// TIA Portal project "BİTİRMEEESON" (V19)

(* hardware
DEVICE "S71500/ET200MP-Station_1"  S7-1500 station
   slot 0: "Profilschiene_0"  6ES7 590-1***0-0AA0
   slot 1: "PLC_1"  CPU 1515-2 PN  6ES7 515-2AM00-0AB0  V1.8
      slot 3: "CPU-Display_1"  6ES7591-1BA00-0AA0
      slot 32768: "PROFINET-Schnittstelle_1"  X1
      slot 33024: "PROFINET interface_1"  X2
   slot 2: "AI 8xU/I/RTD/TC ST_1"  AI 8xU/I/RTD/TC ST  6ES7 531-7KF00-0AB0  V2.0
   slot 3: "AI 8xU/I/RTD/TC ST_2"  AI 8xU/I/RTD/TC ST  6ES7 531-7KF00-0AB0  V2.0
   slot 4: "AI 8xU/I/RTD/TC ST_3"  AI 8xU/I/RTD/TC ST  6ES7 531-7KF00-0AB0  V2.0
   slot 5: "AI 8xU/I/RTD/TC ST_4"  AI 8xU/I/RTD/TC ST  6ES7 531-7KF00-0AB0  V2.0
   slot 6: "DI 16x24VDC BA_1"  DI 16x24VDC BA  6ES7 521-1BH10-0AA0  V1.0
*)

// ===== PLC "PLC_1"  CPU 1515-2 PN =====

VAR_GLOBAL   // PLC tag table "Standard-Variablentabelle"
   "Start_System" AT %I0.0 : Bool;
   "Stop_System" AT %I0.1 : Bool;
   "EmergencyStop" AT %I0.2 : Bool;
   "System" AT %M0.0 : Bool;
   "System_Works_Light" AT %Q0.0 : Bool;
   "System_Not_Working_Light" AT %Q0.1 : Bool;
   "Conveyor1" AT %Q0.2 : Bool;
   "Conveyor2" AT %Q0.3 : Bool;
   "Conveyor3" AT %Q0.4 : Bool;
   "Conveyor4" AT %Q0.5 : Bool;
   "Conveyor5" AT %Q0.6 : Bool;
   "Conveyor6" AT %Q0.7 : Bool;
   "Object_is_Blue" AT %I0.3 : Bool;
   "Object_is_Green" AT %I0.4 : Bool;
   "Blue_So_Left" AT %Q1.0 : Bool;
   "Green_So_Right" AT %Q1.1 : Bool;
   "Mixing_Machine" AT %Q1.2 : Bool;
   "First_Blue_Sensor" AT %I0.5 : Bool;
   "BlueProductConveyor" AT %Q1.3 : Bool;
   "BlueCapConveyor" AT %Q1.4 : Bool;
   "BlueReadyProductConveyor" AT %Q1.5 : Bool;
   "Blue_Product_Sensor" AT %I0.6 : Bool;
   "Blue_Cap_Sensor" AT %I0.7 : Bool;
   "Blue_Product_Positioner" AT %Q1.6 : Bool;
   "Blue_Cap_Positioner" AT %Q1.7 : Bool;
   "Blue_PicknPlace_Grab" AT %Q2.0 : Bool;
   "Blue_PicknPlace_X" AT %Q2.1 : Bool;
   "Blue_PicknPlace_Z" AT %Q2.2 : Bool;
   "Blue_Product_Positioner_Raise" AT %Q2.3 : Bool;
   "Blue_Cap_Emitter" AT %Q2.4 : Bool;
   "Blue_Ready_Sensor" AT %I1.0 : Bool;
   "Blue_Storage_Sensor" AT %I1.1 : Bool;
   "Blue_Roller_Conveyor_1" AT %Q2.5 : Bool;
   "Blue_Roller_Conveyor_2" AT %Q2.6 : Bool;
   "Blue_Roller_Conveyor_3" AT %Q2.7 : Bool;
   "Blue_Roller_Conveyor_4" AT %Q3.0 : Bool;
   "Blue_Roller_Conveyor_5" AT %Q3.1 : Bool;
   "Blue_Roller_Conveyor_6" AT %Q3.2 : Bool;
   "Blue_Ready_Positioner_Clamp" AT %Q3.3 : Bool;
   "Blue_Loading_Conveyor" AT %Q3.4 : Bool;
   "Blue_Box_PicknPlace_X" AT %Q3.5 : Bool;
   "Blue_Box_PicknPlace_Grab" AT %Q3.6 : Bool;
   "Blue_Box_PicknPlace_Z" AT %Q3.7 : Bool;
   "Blue_Conveyor_Blade_1" AT %Q4.0 : Bool;
   "Blue_Conveyor_Blade_2" AT %Q4.1 : Bool;
   "Blue_Box_Emitter" AT %Q4.2 : Bool;
   "Blue_Storage_Start_Button" AT %I1.2 : Bool;
   "Blue_Storage_Stop_Button" AT %I1.3 : Bool;
   "Blue_Storage_Emergency_Button" AT %I1.4 : Bool;
   "Blue_Storage_Start_Button_Main" AT %I1.5 : Bool;
   "Blue_Storage_Stop_Button_Main" AT %I1.6 : Bool;
   "Blue_Storage_Emergency_Button_Main" AT %I1.7 : Bool;
   "Blue_Storage_System" AT %M0.1 : Bool;
   "Blue_Storage_Crane_Left" AT %Q4.3 : Bool;
   "Blue_Storage_Crane_Right" AT %Q4.4 : Bool;
   "Blue_Storage_Crane_Lift" AT %Q4.5 : Bool;
   "Blue_Storage_Start_Button_Light" AT %Q4.6 : Bool;
   "Blue_Storage_Stop_Button_Light" AT %Q4.7 : Bool;
   "Blue_Storage_Start_Button_Main_Light" AT %Q5.0 : Bool;
   "Blue_Storage_Stop_Button_Main_Light" AT %Q5.1 : Bool;
   "Blue_Storage_Reset_Button" AT %I2.0 : Bool;
   "Blue_Storage_Reset_Main_Button" AT %I2.1 : Bool;
   "Blue_Storage_Reset_Button_Light" AT %Q5.2 : Bool;
   "Blue_Storage_Reset_Main_Button_Light" AT %Q5.3 : Bool;
   "Blue_Storage_Crane_Target_Position" AT %QD30 : DInt;
   "Blue_Box_2_Emitter" AT %Q5.4 : Bool;
   "First_Gray_Sensor" AT %I2.2 : Bool;
   "GrayReadyProductConveyor" AT %Q5.5 : Bool;
   "Gray_Cap_Emitter" AT %Q5.6 : Bool;
   "GrayCapConveyor" AT %Q5.7 : Bool;
   "GrayProductConveyor" AT %Q6.0 : Bool;
   "Gray_Product_Sensor" AT %I2.3 : Bool;
   "Gray_Cap_Sensor" AT %I2.4 : Bool;
   "Gray_Product_Positioner" AT %Q6.1 : Bool;
   "Gray_Cap_Positioner" AT %Q6.2 : Bool;
   "Gray_PicknPlace_Grab" AT %Q6.3 : Bool;
   "Gray_PicknPlace_X" AT %Q6.4 : Bool;
   "Gray_PicknPlace_Z" AT %Q6.5 : Bool;
   "Gray_Product_Positioner_Raise" AT %Q6.6 : Bool;
   "Gray_Ready_Sensor" AT %I2.5 : Bool;
   "Gray_Roller_Conveyor_1" AT %Q6.7 : Bool;
   "Gray_Roller_Conveyor_2" AT %Q7.0 : Bool;
   "Gray_Roller_Conveyor_3" AT %Q7.1 : Bool;
   "Gray_Roller_Conveyor_4" AT %Q7.2 : Bool;
   "Gray_Roller_Conveyor_5" AT %Q7.3 : Bool;
   "Gray_Roller_Conveyor_6" AT %Q7.4 : Bool;
   "Gray_Storage_Sensor" AT %I2.6 : Bool;
   "Gray_Loading_Conveyor" AT %Q7.5 : Bool;
   "Gray_Ready_Positioner_Clamp" AT %Q7.6 : Bool;
   "Gray_Box_PicknPlace_X" AT %Q7.7 : Bool;
   "Gray_Box_PicknPlace_Grab" AT %Q8.0 : Bool;
   "Gray_Box_PicknPlace_Z" AT %Q8.1 : Bool;
   "Gray_Box_Emitter" AT %Q8.2 : Bool;
   "Gray_Box_2_Emitter" AT %Q8.3 : Bool;
   "Gray_Conveyor_Blade_1" AT %Q8.4 : Bool;
   "Gray_Conveyor_Blade_2" AT %Q8.5 : Bool;
   "Gray_Storage_Start_Button" AT %I2.7 : Bool;
   "Gray_Storage_Stop_Button" AT %I3.0 : Bool;
   "Gray_Storage_Stop_Button_Main" AT %I3.1 : Bool;
   "Gray_Storage_Emergency_Button" AT %I3.2 : Bool;
   "Gray_Storage_Emergency_Button_Main" AT %I3.3 : Bool;
   "Gray_Storage_System" AT %M0.2 : Bool;
   "Gray_Storage_Start_Button_Main" AT %I3.4 : Bool;
   "Gray_Storage_Reset_Button" AT %I3.5 : Bool;
   "Gray_Storage_Crane_Left" AT %Q8.6 : Bool;
   "Gray_Storage_Reset_Main_Button" AT %I3.6 : Bool;
   "Gray_Storage_Crane_Right" AT %Q8.7 : Bool;
   "Gray_Storage_Crane_Lift" AT %Q9.0 : Bool;
   "Gray_Storage_Start_Button_Light" AT %Q9.1 : Bool;
   "Gray_Storage_Start_Button_Main_Light" AT %Q9.2 : Bool;
   "Gray_Storage_Stop_Button_Light" AT %Q9.3 : Bool;
   "Gray_Storage_Stop_Button_Main_Light" AT %Q9.4 : Bool;
   "Gray_Storage_Reset_Button_Light" AT %Q9.5 : Bool;
   "Gray_Storage_Reset_Main_Button_Light" AT %Q9.6 : Bool;
   "Gray_Storage_Crane_Target_Position" AT %QD34 : DInt;
   "First_Green_Sensor" AT %I3.7 : Bool;
   "GreenReadyProductConveyor" AT %Q9.7 : Bool;
   "Green_Cap_Emitter" AT %Q10.0 : Bool;
   "GreenCapConveyor" AT %Q10.1 : Bool;
   "GreenProductConveyor" AT %Q10.2 : Bool;
   "Green_Product_Positioner" AT %Q10.3 : Bool;
   "Green_Cap_Positioner" AT %Q10.4 : Bool;
   "Green_Product_Sensor" AT %I4.0 : Bool;
   "Green_Cap_Sensor" AT %I4.1 : Bool;
   "Green_PicknPlace_Grab" AT %Q10.5 : Bool;
   "Green_PicknPlace_X" AT %Q10.6 : Bool;
   "Green_PicknPlace_Z" AT %Q10.7 : Bool;
   "Green_Product_Positioner_Raise" AT %Q11.0 : Bool;
   "Green_Ready_Sensor" AT %I4.2 : Bool;
   "Green_Roller_Conveyor_1" AT %Q11.1 : Bool;
   "Green_Roller_Conveyor_2" AT %Q11.2 : Bool;
   "Green_Roller_Conveyor_3" AT %Q11.3 : Bool;
   "Green_Roller_Conveyor_4" AT %Q11.4 : Bool;
   "Green_Roller_Conveyor_5" AT %Q11.5 : Bool;
   "Green_Roller_Conveyor_6" AT %Q11.6 : Bool;
   "Green_Loading_Conveyor" AT %Q11.7 : Bool;
   "Green_Ready_Positioner_Clamp" AT %Q12.0 : Bool;
   "Green_Box_PicknPlace_X" AT %Q12.1 : Bool;
   "Green_Box_PicknPlace_Grab" AT %Q12.2 : Bool;
   "Green_Box_PicknPlace_Z" AT %Q12.3 : Bool;
   "Green_Conveyor_Blade_1" AT %Q12.4 : Bool;
   "Green_Conveyor_Blade_2" AT %Q12.5 : Bool;
   "Green_Box_Emitter" AT %Q12.6 : Bool;
   "Green_Box_2_Emitter" AT %Q12.7 : Bool;
   "Green_Storage_System" AT %M0.3 : Bool;
   "Green_Storage_Start_Button" AT %I4.3 : Bool;
   "Green_Storage_Stop_Button" AT %I4.4 : Bool;
   "Green_Storage_Stop_Button_Main" AT %I4.5 : Bool;
   "Green_Storage_Emergency_Button" AT %I4.6 : Bool;
   "Green_Storage_Emergency_Button_Main" AT %I4.7 : Bool;
   "Green_Storage_Start_Button_Main" AT %I5.0 : Bool;
   "Green_Storage_Reset_Button" AT %I5.1 : Bool;
   "Green_Storage_Reset_Main_Button" AT %I5.2 : Bool;
   "Green_Storage_Crane_Left" AT %Q13.0 : Bool;
   "Green_Storage_Crane_Right" AT %Q13.1 : Bool;
   "Green_Storage_Crane_Lift" AT %Q13.2 : Bool;
   "Green_Storage_Start_Button_Light" AT %Q13.3 : Bool;
   "Green_Storage_Start_Button_Main_Light" AT %Q13.4 : Bool;
   "Green_Storage_Stop_Button_Light" AT %Q13.5 : Bool;
   "Green_Storage_Stop_Button_Main_Light" AT %Q13.6 : Bool;
   "Green_Storage_Reset_Button_Light" AT %Q13.7 : Bool;
   "Green_Storage_Reset_Main_Button_Light" AT %Q14.0 : Bool;
   "Green_Storage_Sensor" AT %I5.3 : Bool;
   "Green_Storage_Crane_Target_Position" AT %QD38 : DInt;
   "MixingCorrectorSensor" AT %I5.4 : Bool;
   "BlueRawEmitter" AT %Q14.1 : Bool;
   "GreenRawEmitter" AT %Q14.2 : Bool;
   "GrayRawEmitter" AT %Q14.3 : Bool;
   "Mixing_Clamp" AT %Q14.4 : Bool;
   "Mixing_Raise" AT %Q14.5 : Bool;
   "Blue_Fill_Valve" AT %QD42 : Real;
   "Blue_Level_Meter" AT %ID30 : DWord;
   "Blue_Liquid_Level" AT %QD56 : DWord;
   "Blue_Norm" AT %MD5 : DWord;
   "Gray_Fill_Valve" AT %QD46 : DWord;
   "Gray_Level_Meter" AT %ID34 : DWord;
   "Gray_Liquid_Level" AT %QD60 : DWord;
   "Gray_Norm" AT %MD6 : DWord;
   "Green_Fill_Valve" AT %QD50 : DWord;
   "Green_Level_Meter" AT %ID38 : DWord;
   "Green_Liquid_Level" AT %QD64 : DWord;
   "Green_Norm" AT %MD7 : DWord;
   "Blue" AT %MW100 : Int;
   "Blue_PID_Flag" AT %M1.0 : Bool;
   "Green_PID_Flag" AT %M1.1 : Bool;
   "Gray_PID_Flag" AT %M1.2 : Bool;
   "Gray" AT %MW104 : Int;
   "Green" AT %MW106 : Int;
   "Blue_Blade_Tank" AT %Q15.2 : Bool;
   "Green_Blade_Tank" AT %Q15.3 : Bool;
   "Gray_Blade_Tank" AT %Q15.4 : Bool;
   "Blue_Base_Vision" AT %I5.5 : Bool;
   "Green_Base_Vision" AT %I5.6 : Bool;
   "Gray_Base_Vision" AT %I5.7 : Bool;
   "BlueDischarge" AT %QD54 : DWord;
   "GreenDischarge" AT %QD58 : DWord;
   "EmitterCycle" AT %M0.4 : Bool;
   "EmittableSituation" AT %M0.5 : Bool;
   "GreenEmit" AT %M0.6 : Bool;
   "GrayEmit" AT %M0.7 : Bool;
   "Conveyor 7" AT %Q14.6 : Bool;
   "Conveyor 8" AT %Q14.7 : Bool;
   "Conveyor 9" AT %Q15.0 : Bool;
   "Conveyor 10" AT %Q15.1 : Bool;
   "Conveyor 11" AT %Q15.5 : Bool;
   "Conveyor 12" AT %Q15.6 : Bool;
   "Conveyor 13" AT %Q15.7 : Bool;
END_VAR

DATA_BLOCK "BrandNewFill_DB"   // DB1
{ S7_Optimized_Access := 'TRUE' }
VERSION : 0.1
// stored: InstanceOfName BrandNewFill
"BrandNewFill"
BEGIN
END_DATA_BLOCK

DATA_BLOCK "Blue_PickPlace_DB"   // DB3
{ S7_Optimized_Access := 'TRUE' }
VERSION : 0.1
// stored: InstanceOfName Blue_PickPlace
"Blue_PickPlace"
BEGIN
END_DATA_BLOCK

DATA_BLOCK "Blue_Storage_Line_DB"   // DB4
{ S7_Optimized_Access := 'TRUE' }
VERSION : 0.1
// stored: InstanceOfName Blue_Storage_Line
"Blue_Storage_Line"
BEGIN
END_DATA_BLOCK

DATA_BLOCK "Blue_Store_DB"   // DB5
{ S7_Optimized_Access := 'TRUE' }
VERSION : 0.1
// stored: InstanceOfName Blue_Store
"Blue_Store"
BEGIN
END_DATA_BLOCK

DATA_BLOCK "Gray_PickPlace_DB"   // DB6
{ S7_Optimized_Access := 'TRUE' }
VERSION : 0.1
// stored: InstanceOfName Gray_PickPlace
"Gray_PickPlace"
BEGIN
END_DATA_BLOCK

DATA_BLOCK "Gray_Storage_Line_DB"   // DB7
{ S7_Optimized_Access := 'TRUE' }
VERSION : 0.1
// stored: InstanceOfName Gray_Storage_Line
"Gray_Storage_Line"
BEGIN
END_DATA_BLOCK

DATA_BLOCK "Gray_Store_DB"   // DB8
{ S7_Optimized_Access := 'TRUE' }
VERSION : 0.1
// stored: InstanceOfName Gray_Store
"Gray_Store"
BEGIN
END_DATA_BLOCK

DATA_BLOCK "Green_PickPlace_DB"   // DB9
{ S7_Optimized_Access := 'TRUE' }
VERSION : 0.1
// stored: InstanceOfName Green_PickPlace
"Green_PickPlace"
BEGIN
END_DATA_BLOCK

DATA_BLOCK "Green_Storage_Line_DB"   // DB10
{ S7_Optimized_Access := 'TRUE' }
VERSION : 0.1
// stored: InstanceOfName Green_Storage_Line
"Green_Storage_Line"
BEGIN
END_DATA_BLOCK

DATA_BLOCK "Green_Store_DB"   // DB11
{ S7_Optimized_Access := 'TRUE' }
VERSION : 0.1
// stored: InstanceOfName Green_Store
"Green_Store"
BEGIN
END_DATA_BLOCK

DATA_BLOCK "MixingCorrector_DB"   // DB108
{ S7_Optimized_Access := 'TRUE' }
VERSION : 0.1
// stored: InstanceOfName MixingCorrector
"MixingCorrector"
BEGIN
END_DATA_BLOCK

// folder: System blocks/Program resources

DATA_BLOCK "TP_BLUEBLADE"   // DB12
{ S7_Optimized_Access := 'TRUE' }
AUTHOR : Simatic
FAMILY : IEC
NAME : IEC_TMR
VERSION : 1.0
// stored: InstanceOfName IEC_TIMER
"IEC_TIMER"
BEGIN
END_DATA_BLOCK

DATA_BLOCK "Blue_Pick&Place"   // DB13
{ S7_Optimized_Access := 'TRUE' }
AUTHOR : Simatic
FAMILY : IEC
NAME : IEC_TMR
VERSION : 1.0
// stored: InstanceOfName IEC_TIMER
"IEC_TIMER"
BEGIN
END_DATA_BLOCK

DATA_BLOCK "Blue_Pick&Place_Grab"   // DB14
{ S7_Optimized_Access := 'TRUE' }
AUTHOR : Simatic
FAMILY : IEC
NAME : IEC_TMR
VERSION : 1.0
// stored: InstanceOfName IEC_TIMER
"IEC_TIMER"
BEGIN
END_DATA_BLOCK

DATA_BLOCK "Blue_Pick&Place_TON_X"   // DB15
{ S7_Optimized_Access := 'TRUE' }
AUTHOR : Simatic
FAMILY : IEC
NAME : IEC_TMR
VERSION : 1.0
// stored: InstanceOfName IEC_TIMER
"IEC_TIMER"
BEGIN
END_DATA_BLOCK

DATA_BLOCK "Blue_Pick&Place_TP_X"   // DB16
{ S7_Optimized_Access := 'TRUE' }
AUTHOR : Simatic
FAMILY : IEC
NAME : IEC_TMR
VERSION : 1.0
// stored: InstanceOfName IEC_TIMER
"IEC_TIMER"
BEGIN
END_DATA_BLOCK

DATA_BLOCK "Blue_Pick&Place_TON_Z1"   // DB17
{ S7_Optimized_Access := 'TRUE' }
AUTHOR : Simatic
FAMILY : IEC
NAME : IEC_TMR
VERSION : 1.0
// stored: InstanceOfName IEC_TIMER
"IEC_TIMER"
BEGIN
END_DATA_BLOCK

DATA_BLOCK "Blue_Pick&PlaceZ2"   // DB18
{ S7_Optimized_Access := 'TRUE' }
AUTHOR : Simatic
FAMILY : IEC
NAME : IEC_TMR
VERSION : 1.0
// stored: InstanceOfName IEC_TIMER
"IEC_TIMER"
BEGIN
END_DATA_BLOCK

DATA_BLOCK "Blue_Pick&PlaceZ3"   // DB19
{ S7_Optimized_Access := 'TRUE' }
AUTHOR : Simatic
FAMILY : IEC
NAME : IEC_TMR
VERSION : 1.0
// stored: InstanceOfName IEC_TIMER
"IEC_TIMER"
BEGIN
END_DATA_BLOCK

DATA_BLOCK "Blue_Raise"   // DB20
{ S7_Optimized_Access := 'TRUE' }
AUTHOR : Simatic
FAMILY : IEC
NAME : IEC_TMR
VERSION : 1.0
// stored: InstanceOfName IEC_TIMER
"IEC_TIMER"
BEGIN
END_DATA_BLOCK

DATA_BLOCK "Blue_Box_Pick&Place"   // DB21
{ S7_Optimized_Access := 'TRUE' }
AUTHOR : Simatic
FAMILY : IEC
NAME : IEC_TMR
VERSION : 1.0
// stored: InstanceOfName IEC_TIMER
"IEC_TIMER"
BEGIN
END_DATA_BLOCK

DATA_BLOCK "Blue_Box_Pick&Place_TON_Grab"   // DB22
{ S7_Optimized_Access := 'TRUE' }
AUTHOR : Simatic
FAMILY : IEC
NAME : IEC_TMR
VERSION : 1.0
// stored: InstanceOfName IEC_TIMER
"IEC_TIMER"
BEGIN
END_DATA_BLOCK

DATA_BLOCK "GrayConveyor"   // DB23
{ S7_Optimized_Access := 'TRUE' }
AUTHOR : Simatic
FAMILY : IEC
NAME : IEC_TMR
VERSION : 1.0
// stored: InstanceOfName IEC_TIMER
"IEC_TIMER"
BEGIN
END_DATA_BLOCK

DATA_BLOCK "Gray_Pick&Place"   // DB24
{ S7_Optimized_Access := 'TRUE' }
AUTHOR : Simatic
FAMILY : IEC
NAME : IEC_TMR
VERSION : 1.0
// stored: InstanceOfName IEC_TIMER
"IEC_TIMER"
BEGIN
END_DATA_BLOCK

DATA_BLOCK "Blue_Storage_Set_TP"   // DB25
{ S7_Optimized_Access := 'TRUE' }
AUTHOR : Simatic
FAMILY : IEC
NAME : IEC_TMR
VERSION : 1.0
// stored: InstanceOfName IEC_TIMER
"IEC_TIMER"
BEGIN
END_DATA_BLOCK

DATA_BLOCK "Blue_Storage_CTU"   // DB26
{ S7_Optimized_Access := 'TRUE' }
AUTHOR : Simatic
FAMILY : IEC
NAME : CNTR
VERSION : 1.0
// stored: InstanceOfName IEC_COUNTER
"IEC_COUNTER"
BEGIN
END_DATA_BLOCK

DATA_BLOCK "Blue_Storage_CTU_Reset_TON"   // DB27
{ S7_Optimized_Access := 'TRUE' }
AUTHOR : Simatic
FAMILY : IEC
NAME : IEC_TMR
VERSION : 1.0
// stored: InstanceOfName IEC_TIMER
"IEC_TIMER"
BEGIN
END_DATA_BLOCK

DATA_BLOCK "Gray_Pick&Place_Grab"   // DB28
{ S7_Optimized_Access := 'TRUE' }
AUTHOR : Simatic
FAMILY : IEC
NAME : IEC_TMR
VERSION : 1.0
// stored: InstanceOfName IEC_TIMER
"IEC_TIMER"
BEGIN
END_DATA_BLOCK

DATA_BLOCK "Gray_Pick&Place_TON_X"   // DB29
{ S7_Optimized_Access := 'TRUE' }
AUTHOR : Simatic
FAMILY : IEC
NAME : IEC_TMR
VERSION : 1.0
// stored: InstanceOfName IEC_TIMER
"IEC_TIMER"
BEGIN
END_DATA_BLOCK

DATA_BLOCK "Blue_Box_Pick&Place_TON_Z1"   // DB30
{ S7_Optimized_Access := 'TRUE' }
AUTHOR : Simatic
FAMILY : IEC
NAME : IEC_TMR
VERSION : 1.0
// stored: InstanceOfName IEC_TIMER
"IEC_TIMER"
BEGIN
END_DATA_BLOCK

DATA_BLOCK "Blue_Box_Pick&Place_TP_Z"   // DB31
{ S7_Optimized_Access := 'TRUE' }
AUTHOR : Simatic
FAMILY : IEC
NAME : IEC_TMR
VERSION : 1.0
// stored: InstanceOfName IEC_TIMER
"IEC_TIMER"
BEGIN
END_DATA_BLOCK

DATA_BLOCK "Blue_Box_Pick&Place_TON_Z2"   // DB32
{ S7_Optimized_Access := 'TRUE' }
AUTHOR : Simatic
FAMILY : IEC
NAME : IEC_TMR
VERSION : 1.0
// stored: InstanceOfName IEC_TIMER
"IEC_TIMER"
BEGIN
END_DATA_BLOCK

DATA_BLOCK "Blue_Box_Pick&Place_TON_Z3"   // DB33
{ S7_Optimized_Access := 'TRUE' }
AUTHOR : Simatic
FAMILY : IEC
NAME : IEC_TMR
VERSION : 1.0
// stored: InstanceOfName IEC_TIMER
"IEC_TIMER"
BEGIN
END_DATA_BLOCK

DATA_BLOCK "Gray_Pick&Place_TP_X"   // DB34
{ S7_Optimized_Access := 'TRUE' }
AUTHOR : Simatic
FAMILY : IEC
NAME : IEC_TMR
VERSION : 1.0
// stored: InstanceOfName IEC_TIMER
"IEC_TIMER"
BEGIN
END_DATA_BLOCK

DATA_BLOCK "Blue_Box_Pick&Place_X"   // DB35
{ S7_Optimized_Access := 'TRUE' }
AUTHOR : Simatic
FAMILY : IEC
NAME : IEC_TMR
VERSION : 1.0
// stored: InstanceOfName IEC_TIMER
"IEC_TIMER"
BEGIN
END_DATA_BLOCK

DATA_BLOCK "Blue_Box_Pick&Place_TP_Grab"   // DB36
{ S7_Optimized_Access := 'TRUE' }
AUTHOR : Simatic
FAMILY : IEC
NAME : IEC_TMR
VERSION : 1.0
// stored: InstanceOfName IEC_TIMER
"IEC_TIMER"
BEGIN
END_DATA_BLOCK

DATA_BLOCK "Gray_Pick&Place_TON_Z1"   // DB37
{ S7_Optimized_Access := 'TRUE' }
AUTHOR : Simatic
FAMILY : IEC
NAME : IEC_TMR
VERSION : 1.0
// stored: InstanceOfName IEC_TIMER
"IEC_TIMER"
BEGIN
END_DATA_BLOCK

DATA_BLOCK "Gray_Pick&PlaceZ2"   // DB38
{ S7_Optimized_Access := 'TRUE' }
AUTHOR : Simatic
FAMILY : IEC
NAME : IEC_TMR
VERSION : 1.0
// stored: InstanceOfName IEC_TIMER
"IEC_TIMER"
BEGIN
END_DATA_BLOCK

DATA_BLOCK "Gray_Pick&PlaceZ3"   // DB39
{ S7_Optimized_Access := 'TRUE' }
AUTHOR : Simatic
FAMILY : IEC
NAME : IEC_TMR
VERSION : 1.0
// stored: InstanceOfName IEC_TIMER
"IEC_TIMER"
BEGIN
END_DATA_BLOCK

DATA_BLOCK "Gray_Raise"   // DB40
{ S7_Optimized_Access := 'TRUE' }
AUTHOR : Simatic
FAMILY : IEC
NAME : IEC_TMR
VERSION : 1.0
// stored: InstanceOfName IEC_TIMER
"IEC_TIMER"
BEGIN
END_DATA_BLOCK

DATA_BLOCK "GrayCapConvey"   // DB41
{ S7_Optimized_Access := 'TRUE' }
AUTHOR : Simatic
FAMILY : IEC
NAME : IEC_TMR
VERSION : 1.0
// stored: InstanceOfName IEC_TIMER
"IEC_TIMER"
BEGIN
END_DATA_BLOCK

DATA_BLOCK "Gray_Box_Pick&Place"   // DB42
{ S7_Optimized_Access := 'TRUE' }
AUTHOR : Simatic
FAMILY : IEC
NAME : IEC_TMR
VERSION : 1.0
// stored: InstanceOfName IEC_TIMER
"IEC_TIMER"
BEGIN
END_DATA_BLOCK

DATA_BLOCK "Gray_Box_Pick&Place_X"   // DB43
{ S7_Optimized_Access := 'TRUE' }
AUTHOR : Simatic
FAMILY : IEC
NAME : IEC_TMR
VERSION : 1.0
// stored: InstanceOfName IEC_TIMER
"IEC_TIMER"
BEGIN
END_DATA_BLOCK

DATA_BLOCK "Gray_Box_Pick&Place_TON_Grab"   // DB44
{ S7_Optimized_Access := 'TRUE' }
AUTHOR : Simatic
FAMILY : IEC
NAME : IEC_TMR
VERSION : 1.0
// stored: InstanceOfName IEC_TIMER
"IEC_TIMER"
BEGIN
END_DATA_BLOCK

DATA_BLOCK "Gray_Box_Pick&Place_TP_Grab"   // DB45
{ S7_Optimized_Access := 'TRUE' }
AUTHOR : Simatic
FAMILY : IEC
NAME : IEC_TMR
VERSION : 1.0
// stored: InstanceOfName IEC_TIMER
"IEC_TIMER"
BEGIN
END_DATA_BLOCK

DATA_BLOCK "Gray_Box_Pick&Place_TON_Z1"   // DB46
{ S7_Optimized_Access := 'TRUE' }
AUTHOR : Simatic
FAMILY : IEC
NAME : IEC_TMR
VERSION : 1.0
// stored: InstanceOfName IEC_TIMER
"IEC_TIMER"
BEGIN
END_DATA_BLOCK

DATA_BLOCK "Gray_Box_Pick&Place_TP_Z"   // DB47
{ S7_Optimized_Access := 'TRUE' }
AUTHOR : Simatic
FAMILY : IEC
NAME : IEC_TMR
VERSION : 1.0
// stored: InstanceOfName IEC_TIMER
"IEC_TIMER"
BEGIN
END_DATA_BLOCK

DATA_BLOCK "Gray_Box_Pick&Place_TON_Z2"   // DB48
{ S7_Optimized_Access := 'TRUE' }
AUTHOR : Simatic
FAMILY : IEC
NAME : IEC_TMR
VERSION : 1.0
// stored: InstanceOfName IEC_TIMER
"IEC_TIMER"
BEGIN
END_DATA_BLOCK

DATA_BLOCK "Gray_Box_Pick&Place_TON_Z3"   // DB49
{ S7_Optimized_Access := 'TRUE' }
AUTHOR : Simatic
FAMILY : IEC
NAME : IEC_TMR
VERSION : 1.0
// stored: InstanceOfName IEC_TIMER
"IEC_TIMER"
BEGIN
END_DATA_BLOCK

DATA_BLOCK "Gray_Box_XTU"   // DB50
{ S7_Optimized_Access := 'TRUE' }
AUTHOR : Simatic
FAMILY : IEC
NAME : CNTR
VERSION : 1.0
// stored: InstanceOfName IEC_COUNTER
"IEC_COUNTER"
BEGIN
END_DATA_BLOCK

DATA_BLOCK "Gray_Box_TON"   // DB51
{ S7_Optimized_Access := 'TRUE' }
AUTHOR : Simatic
FAMILY : IEC
NAME : IEC_TMR
VERSION : 1.0
// stored: InstanceOfName IEC_TIMER
"IEC_TIMER"
BEGIN
END_DATA_BLOCK

DATA_BLOCK "BlueConveyor"   // DB52
{ S7_Optimized_Access := 'TRUE' }
AUTHOR : Simatic
FAMILY : IEC
NAME : IEC_TMR
VERSION : 1.0
// stored: InstanceOfName IEC_TIMER
"IEC_TIMER"
BEGIN
END_DATA_BLOCK

DATA_BLOCK "BlueCapConvey"   // DB53
{ S7_Optimized_Access := 'TRUE' }
AUTHOR : Simatic
FAMILY : IEC
NAME : IEC_TMR
VERSION : 1.0
// stored: InstanceOfName IEC_TIMER
"IEC_TIMER"
BEGIN
END_DATA_BLOCK

DATA_BLOCK "Blue_Box_TON"   // DB54
{ S7_Optimized_Access := 'TRUE' }
AUTHOR : Simatic
FAMILY : IEC
NAME : IEC_TMR
VERSION : 1.0
// stored: InstanceOfName IEC_TIMER
"IEC_TIMER"
BEGIN
END_DATA_BLOCK

DATA_BLOCK "Blue_Box_XTU"   // DB55
{ S7_Optimized_Access := 'TRUE' }
AUTHOR : Simatic
FAMILY : IEC
NAME : CNTR
VERSION : 1.0
// stored: InstanceOfName IEC_COUNTER
"IEC_COUNTER"
BEGIN
END_DATA_BLOCK

DATA_BLOCK "Blue_Box_TP"   // DB56
{ S7_Optimized_Access := 'TRUE' }
AUTHOR : Simatic
FAMILY : IEC
NAME : IEC_TMR
VERSION : 1.0
// stored: InstanceOfName IEC_TIMER
"IEC_TIMER"
BEGIN
END_DATA_BLOCK

DATA_BLOCK "Gray_Box_TP"   // DB57
{ S7_Optimized_Access := 'TRUE' }
AUTHOR : Simatic
FAMILY : IEC
NAME : IEC_TMR
VERSION : 1.0
// stored: InstanceOfName IEC_TIMER
"IEC_TIMER"
BEGIN
END_DATA_BLOCK

DATA_BLOCK "Gray_Storage_CTU"   // DB58
{ S7_Optimized_Access := 'TRUE' }
AUTHOR : Simatic
FAMILY : IEC
NAME : CNTR
VERSION : 1.0
// stored: InstanceOfName IEC_COUNTER
"IEC_COUNTER"
BEGIN
END_DATA_BLOCK

DATA_BLOCK "Gray_Storage_CTU_Reset_TON"   // DB59
{ S7_Optimized_Access := 'TRUE' }
AUTHOR : Simatic
FAMILY : IEC
NAME : IEC_TMR
VERSION : 1.0
// stored: InstanceOfName IEC_TIMER
"IEC_TIMER"
BEGIN
END_DATA_BLOCK

DATA_BLOCK "Gray_Storage_Set_TP"   // DB60
{ S7_Optimized_Access := 'TRUE' }
AUTHOR : Simatic
FAMILY : IEC
NAME : IEC_TMR
VERSION : 1.0
// stored: InstanceOfName IEC_TIMER
"IEC_TIMER"
BEGIN
END_DATA_BLOCK

DATA_BLOCK "Gray_Storage_Crane_Left_Set"   // DB61
{ S7_Optimized_Access := 'TRUE' }
AUTHOR : Simatic
FAMILY : IEC
NAME : IEC_TMR
VERSION : 1.0
// stored: InstanceOfName IEC_TIMER
"IEC_TIMER"
BEGIN
END_DATA_BLOCK

DATA_BLOCK "Gray_Stacker_Crane_Right_Set_TON"   // DB62
{ S7_Optimized_Access := 'TRUE' }
AUTHOR : Simatic
FAMILY : IEC
NAME : IEC_TMR
VERSION : 1.0
// stored: InstanceOfName IEC_TIMER
"IEC_TIMER"
BEGIN
END_DATA_BLOCK

DATA_BLOCK "Gray_Storage_Crane_Right_Set_TP"   // DB63
{ S7_Optimized_Access := 'TRUE' }
AUTHOR : Simatic
FAMILY : IEC
NAME : IEC_TMR
VERSION : 1.0
// stored: InstanceOfName IEC_TIMER
"IEC_TIMER"
BEGIN
END_DATA_BLOCK

DATA_BLOCK "Gray_Storage_Crane_Lift_TON"   // DB64
{ S7_Optimized_Access := 'TRUE' }
AUTHOR : Simatic
FAMILY : IEC
NAME : IEC_TMR
VERSION : 1.0
// stored: InstanceOfName IEC_TIMER
"IEC_TIMER"
BEGIN
END_DATA_BLOCK

DATA_BLOCK "Gray_Storage_Crane_Lift_TP"   // DB65
{ S7_Optimized_Access := 'TRUE' }
AUTHOR : Simatic
FAMILY : IEC
NAME : IEC_TMR
VERSION : 1.0
// stored: InstanceOfName IEC_TIMER
"IEC_TIMER"
BEGIN
END_DATA_BLOCK

DATA_BLOCK "Gray_Storage_Position_Set"   // DB66
{ S7_Optimized_Access := 'TRUE' }
AUTHOR : Simatic
FAMILY : IEC
NAME : IEC_TMR
VERSION : 1.0
// stored: InstanceOfName IEC_TIMER
"IEC_TIMER"
BEGIN
END_DATA_BLOCK

DATA_BLOCK "Gray_Storage_Position_Reset"   // DB67
{ S7_Optimized_Access := 'TRUE' }
AUTHOR : Simatic
FAMILY : IEC
NAME : IEC_TMR
VERSION : 1.0
// stored: InstanceOfName IEC_TIMER
"IEC_TIMER"
BEGIN
END_DATA_BLOCK

DATA_BLOCK "GreenConveyor"   // DB68
{ S7_Optimized_Access := 'TRUE' }
AUTHOR : Simatic
FAMILY : IEC
NAME : IEC_TMR
VERSION : 1.0
// stored: InstanceOfName IEC_TIMER
"IEC_TIMER"
BEGIN
END_DATA_BLOCK

DATA_BLOCK "Blue_Storage_Crane_Left_Set"   // DB69
{ S7_Optimized_Access := 'TRUE' }
AUTHOR : Simatic
FAMILY : IEC
NAME : IEC_TMR
VERSION : 1.0
// stored: InstanceOfName IEC_TIMER
"IEC_TIMER"
BEGIN
END_DATA_BLOCK

DATA_BLOCK "Green_Pick&Place"   // DB70
{ S7_Optimized_Access := 'TRUE' }
AUTHOR : Simatic
FAMILY : IEC
NAME : IEC_TMR
VERSION : 1.0
// stored: InstanceOfName IEC_TIMER
"IEC_TIMER"
BEGIN
END_DATA_BLOCK

DATA_BLOCK "Blue_Stacker_Crane_Right_Set_TON"   // DB71
{ S7_Optimized_Access := 'TRUE' }
AUTHOR : Simatic
FAMILY : IEC
NAME : IEC_TMR
VERSION : 1.0
// stored: InstanceOfName IEC_TIMER
"IEC_TIMER"
BEGIN
END_DATA_BLOCK

DATA_BLOCK "Blue_Storage_Crane_Right_Set_TP"   // DB72
{ S7_Optimized_Access := 'TRUE' }
AUTHOR : Simatic
FAMILY : IEC
NAME : IEC_TMR
VERSION : 1.0
// stored: InstanceOfName IEC_TIMER
"IEC_TIMER"
BEGIN
END_DATA_BLOCK

DATA_BLOCK "Blue_Storage_Crane_Lift_TON"   // DB73
{ S7_Optimized_Access := 'TRUE' }
AUTHOR : Simatic
FAMILY : IEC
NAME : IEC_TMR
VERSION : 1.0
// stored: InstanceOfName IEC_TIMER
"IEC_TIMER"
BEGIN
END_DATA_BLOCK

DATA_BLOCK "Blue_Storage_Crane_Lift_TP"   // DB74
{ S7_Optimized_Access := 'TRUE' }
AUTHOR : Simatic
FAMILY : IEC
NAME : IEC_TMR
VERSION : 1.0
// stored: InstanceOfName IEC_TIMER
"IEC_TIMER"
BEGIN
END_DATA_BLOCK

DATA_BLOCK "Blue_Storage_Position_Set"   // DB75
{ S7_Optimized_Access := 'TRUE' }
AUTHOR : Simatic
FAMILY : IEC
NAME : IEC_TMR
VERSION : 1.0
// stored: InstanceOfName IEC_TIMER
"IEC_TIMER"
BEGIN
END_DATA_BLOCK

DATA_BLOCK "Blue_Storage_Position_Reset"   // DB76
{ S7_Optimized_Access := 'TRUE' }
AUTHOR : Simatic
FAMILY : IEC
NAME : IEC_TMR
VERSION : 1.0
// stored: InstanceOfName IEC_TIMER
"IEC_TIMER"
BEGIN
END_DATA_BLOCK

DATA_BLOCK "Green_Pick&Place_Grab"   // DB77
{ S7_Optimized_Access := 'TRUE' }
AUTHOR : Simatic
FAMILY : IEC
NAME : IEC_TMR
VERSION : 1.0
// stored: InstanceOfName IEC_TIMER
"IEC_TIMER"
BEGIN
END_DATA_BLOCK

DATA_BLOCK "Green_Pick&Place_TON_X"   // DB78
{ S7_Optimized_Access := 'TRUE' }
AUTHOR : Simatic
FAMILY : IEC
NAME : IEC_TMR
VERSION : 1.0
// stored: InstanceOfName IEC_TIMER
"IEC_TIMER"
BEGIN
END_DATA_BLOCK

DATA_BLOCK "Green_Pick&Place_TP_X"   // DB79
{ S7_Optimized_Access := 'TRUE' }
AUTHOR : Simatic
FAMILY : IEC
NAME : IEC_TMR
VERSION : 1.0
// stored: InstanceOfName IEC_TIMER
"IEC_TIMER"
BEGIN
END_DATA_BLOCK

DATA_BLOCK "Green_Pick&Place_TON_Z1"   // DB80
{ S7_Optimized_Access := 'TRUE' }
AUTHOR : Simatic
FAMILY : IEC
NAME : IEC_TMR
VERSION : 1.0
// stored: InstanceOfName IEC_TIMER
"IEC_TIMER"
BEGIN
END_DATA_BLOCK

DATA_BLOCK "Green_Pick&PlaceZ2"   // DB81
{ S7_Optimized_Access := 'TRUE' }
AUTHOR : Simatic
FAMILY : IEC
NAME : IEC_TMR
VERSION : 1.0
// stored: InstanceOfName IEC_TIMER
"IEC_TIMER"
BEGIN
END_DATA_BLOCK

DATA_BLOCK "Green_Pick&PlaceZ3"   // DB82
{ S7_Optimized_Access := 'TRUE' }
AUTHOR : Simatic
FAMILY : IEC
NAME : IEC_TMR
VERSION : 1.0
// stored: InstanceOfName IEC_TIMER
"IEC_TIMER"
BEGIN
END_DATA_BLOCK

DATA_BLOCK "Green_Raise"   // DB83
{ S7_Optimized_Access := 'TRUE' }
AUTHOR : Simatic
FAMILY : IEC
NAME : IEC_TMR
VERSION : 1.0
// stored: InstanceOfName IEC_TIMER
"IEC_TIMER"
BEGIN
END_DATA_BLOCK

DATA_BLOCK "GreenCapConvey"   // DB84
{ S7_Optimized_Access := 'TRUE' }
AUTHOR : Simatic
FAMILY : IEC
NAME : IEC_TMR
VERSION : 1.0
// stored: InstanceOfName IEC_TIMER
"IEC_TIMER"
BEGIN
END_DATA_BLOCK

DATA_BLOCK "Green_Box_Pick&Place"   // DB85
{ S7_Optimized_Access := 'TRUE' }
AUTHOR : Simatic
FAMILY : IEC
NAME : IEC_TMR
VERSION : 1.0
// stored: InstanceOfName IEC_TIMER
"IEC_TIMER"
BEGIN
END_DATA_BLOCK

DATA_BLOCK "Green_Box_Pick&Place_X"   // DB86
{ S7_Optimized_Access := 'TRUE' }
AUTHOR : Simatic
FAMILY : IEC
NAME : IEC_TMR
VERSION : 1.0
// stored: InstanceOfName IEC_TIMER
"IEC_TIMER"
BEGIN
END_DATA_BLOCK

DATA_BLOCK "Green_Box_Pick&Place_TON_Grab"   // DB87
{ S7_Optimized_Access := 'TRUE' }
AUTHOR : Simatic
FAMILY : IEC
NAME : IEC_TMR
VERSION : 1.0
// stored: InstanceOfName IEC_TIMER
"IEC_TIMER"
BEGIN
END_DATA_BLOCK

DATA_BLOCK "Green_Box_Pick&Place_TP_Grab"   // DB88
{ S7_Optimized_Access := 'TRUE' }
AUTHOR : Simatic
FAMILY : IEC
NAME : IEC_TMR
VERSION : 1.0
// stored: InstanceOfName IEC_TIMER
"IEC_TIMER"
BEGIN
END_DATA_BLOCK

DATA_BLOCK "Green_Box_Pick&Place_TON_Z1"   // DB89
{ S7_Optimized_Access := 'TRUE' }
AUTHOR : Simatic
FAMILY : IEC
NAME : IEC_TMR
VERSION : 1.0
// stored: InstanceOfName IEC_TIMER
"IEC_TIMER"
BEGIN
END_DATA_BLOCK

DATA_BLOCK "Green_Box_Pick&Place_TP_Z"   // DB90
{ S7_Optimized_Access := 'TRUE' }
AUTHOR : Simatic
FAMILY : IEC
NAME : IEC_TMR
VERSION : 1.0
// stored: InstanceOfName IEC_TIMER
"IEC_TIMER"
BEGIN
END_DATA_BLOCK

DATA_BLOCK "Green_Box_Pick&Place_TON_Z2"   // DB91
{ S7_Optimized_Access := 'TRUE' }
AUTHOR : Simatic
FAMILY : IEC
NAME : IEC_TMR
VERSION : 1.0
// stored: InstanceOfName IEC_TIMER
"IEC_TIMER"
BEGIN
END_DATA_BLOCK

DATA_BLOCK "Green_Box_Pick&Place_TON_Z3"   // DB92
{ S7_Optimized_Access := 'TRUE' }
AUTHOR : Simatic
FAMILY : IEC
NAME : IEC_TMR
VERSION : 1.0
// stored: InstanceOfName IEC_TIMER
"IEC_TIMER"
BEGIN
END_DATA_BLOCK

DATA_BLOCK "Green_Box_XTU"   // DB93
{ S7_Optimized_Access := 'TRUE' }
AUTHOR : Simatic
FAMILY : IEC
NAME : CNTR
VERSION : 1.0
// stored: InstanceOfName IEC_COUNTER
"IEC_COUNTER"
BEGIN
END_DATA_BLOCK

DATA_BLOCK "Green_Box_TON"   // DB94
{ S7_Optimized_Access := 'TRUE' }
AUTHOR : Simatic
FAMILY : IEC
NAME : IEC_TMR
VERSION : 1.0
// stored: InstanceOfName IEC_TIMER
"IEC_TIMER"
BEGIN
END_DATA_BLOCK

DATA_BLOCK "Green_Box_TP"   // DB95
{ S7_Optimized_Access := 'TRUE' }
AUTHOR : Simatic
FAMILY : IEC
NAME : IEC_TMR
VERSION : 1.0
// stored: InstanceOfName IEC_TIMER
"IEC_TIMER"
BEGIN
END_DATA_BLOCK

DATA_BLOCK "Green_Storage_CTU"   // DB96
{ S7_Optimized_Access := 'TRUE' }
AUTHOR : Simatic
FAMILY : IEC
NAME : CNTR
VERSION : 1.0
// stored: InstanceOfName IEC_COUNTER
"IEC_COUNTER"
BEGIN
END_DATA_BLOCK

DATA_BLOCK "Green_Storage_CTU_Reset_TON"   // DB97
{ S7_Optimized_Access := 'TRUE' }
AUTHOR : Simatic
FAMILY : IEC
NAME : IEC_TMR
VERSION : 1.0
// stored: InstanceOfName IEC_TIMER
"IEC_TIMER"
BEGIN
END_DATA_BLOCK

DATA_BLOCK "Green_Storage_Set_TP"   // DB98
{ S7_Optimized_Access := 'TRUE' }
AUTHOR : Simatic
FAMILY : IEC
NAME : IEC_TMR
VERSION : 1.0
// stored: InstanceOfName IEC_TIMER
"IEC_TIMER"
BEGIN
END_DATA_BLOCK

DATA_BLOCK "Green_Storage_Crane_Left_Set"   // DB99
{ S7_Optimized_Access := 'TRUE' }
AUTHOR : Simatic
FAMILY : IEC
NAME : IEC_TMR
VERSION : 1.0
// stored: InstanceOfName IEC_TIMER
"IEC_TIMER"
BEGIN
END_DATA_BLOCK

DATA_BLOCK "Green_Stacker_Crane_Right_Set_TON"   // DB100
{ S7_Optimized_Access := 'TRUE' }
AUTHOR : Simatic
FAMILY : IEC
NAME : IEC_TMR
VERSION : 1.0
// stored: InstanceOfName IEC_TIMER
"IEC_TIMER"
BEGIN
END_DATA_BLOCK

DATA_BLOCK "Green_Storage_Crane_Right_Set_TP"   // DB101
{ S7_Optimized_Access := 'TRUE' }
AUTHOR : Simatic
FAMILY : IEC
NAME : IEC_TMR
VERSION : 1.0
// stored: InstanceOfName IEC_TIMER
"IEC_TIMER"
BEGIN
END_DATA_BLOCK

DATA_BLOCK "Green_Storage_Crane_Lift_TON"   // DB102
{ S7_Optimized_Access := 'TRUE' }
AUTHOR : Simatic
FAMILY : IEC
NAME : IEC_TMR
VERSION : 1.0
// stored: InstanceOfName IEC_TIMER
"IEC_TIMER"
BEGIN
END_DATA_BLOCK

DATA_BLOCK "Green_Storage_Crane_Lift_TP"   // DB103
{ S7_Optimized_Access := 'TRUE' }
AUTHOR : Simatic
FAMILY : IEC
NAME : IEC_TMR
VERSION : 1.0
// stored: InstanceOfName IEC_TIMER
"IEC_TIMER"
BEGIN
END_DATA_BLOCK

DATA_BLOCK "Green_Storage_Position_Set"   // DB104
{ S7_Optimized_Access := 'TRUE' }
AUTHOR : Simatic
FAMILY : IEC
NAME : IEC_TMR
VERSION : 1.0
// stored: InstanceOfName IEC_TIMER
"IEC_TIMER"
BEGIN
END_DATA_BLOCK

DATA_BLOCK "Green_Storage_Position_Reset"   // DB105
{ S7_Optimized_Access := 'TRUE' }
AUTHOR : Simatic
FAMILY : IEC
NAME : IEC_TMR
VERSION : 1.0
// stored: InstanceOfName IEC_TIMER
"IEC_TIMER"
BEGIN
END_DATA_BLOCK

DATA_BLOCK "MixClampTP"   // DB106
{ S7_Optimized_Access := 'TRUE' }
AUTHOR : Simatic
FAMILY : IEC
NAME : IEC_TMR
VERSION : 1.0
// stored: InstanceOfName IEC_TIMER
"IEC_TIMER"
BEGIN
END_DATA_BLOCK

DATA_BLOCK "MixRaiseTP"   // DB107
{ S7_Optimized_Access := 'TRUE' }
AUTHOR : Simatic
FAMILY : IEC
NAME : IEC_TMR
VERSION : 1.0
// stored: InstanceOfName IEC_TIMER
"IEC_TIMER"
BEGIN
END_DATA_BLOCK

DATA_BLOCK "TP_GREEN_BLADE"   // DB109
{ S7_Optimized_Access := 'TRUE' }
AUTHOR : Simatic
FAMILY : IEC
NAME : IEC_TMR
VERSION : 1.0
// stored: InstanceOfName IEC_TIMER
"IEC_TIMER"
BEGIN
END_DATA_BLOCK

DATA_BLOCK "TP_GRAY_BLADE"   // DB110
{ S7_Optimized_Access := 'TRUE' }
AUTHOR : Simatic
FAMILY : IEC
NAME : IEC_TMR
VERSION : 1.0
// stored: InstanceOfName IEC_TIMER
"IEC_TIMER"
BEGIN
END_DATA_BLOCK

DATA_BLOCK "TONGREEN"   // DB111
{ S7_Optimized_Access := 'TRUE' }
AUTHOR : Simatic
FAMILY : IEC
NAME : IEC_TMR
VERSION : 1.0
// stored: InstanceOfName IEC_TIMER
"IEC_TIMER"
BEGIN
END_DATA_BLOCK

DATA_BLOCK "TONGRay"   // DB112
{ S7_Optimized_Access := 'TRUE' }
AUTHOR : Simatic
FAMILY : IEC
NAME : IEC_TMR
VERSION : 1.0
// stored: InstanceOfName IEC_TIMER
"IEC_TIMER"
BEGIN
END_DATA_BLOCK

DATA_BLOCK "TONBLUE"   // DB113
{ S7_Optimized_Access := 'TRUE' }
AUTHOR : Simatic
FAMILY : IEC
NAME : IEC_TMR
VERSION : 1.0
// stored: InstanceOfName IEC_TIMER
"IEC_TIMER"
BEGIN
END_DATA_BLOCK

DATA_BLOCK "StarterTimer"   // DB114
{ S7_Optimized_Access := 'TRUE' }
AUTHOR : Simatic
FAMILY : IEC
NAME : IEC_TMR
VERSION : 1.0
// stored: InstanceOfName IEC_TIMER
"IEC_TIMER"
BEGIN
END_DATA_BLOCK

DATA_BLOCK "InitialTimer"   // DB115
{ S7_Optimized_Access := 'TRUE' }
AUTHOR : Simatic
FAMILY : IEC
NAME : IEC_TMR
VERSION : 1.0
// stored: InstanceOfName IEC_TIMER
"IEC_TIMER"
BEGIN
END_DATA_BLOCK

DATA_BLOCK "TPGREENTP"   // DB116
{ S7_Optimized_Access := 'TRUE' }
AUTHOR : Simatic
FAMILY : IEC
NAME : IEC_TMR
VERSION : 1.0
// stored: InstanceOfName IEC_TIMER
"IEC_TIMER"
BEGIN
END_DATA_BLOCK

DATA_BLOCK "TPGrayTP"   // DB117
{ S7_Optimized_Access := 'TRUE' }
AUTHOR : Simatic
FAMILY : IEC
NAME : IEC_TMR
VERSION : 1.0
// stored: InstanceOfName IEC_TIMER
"IEC_TIMER"
BEGIN
END_DATA_BLOCK

DATA_BLOCK "TPBLUETP"   // DB118
{ S7_Optimized_Access := 'TRUE' }
AUTHOR : Simatic
FAMILY : IEC
NAME : IEC_TMR
VERSION : 1.0
// stored: InstanceOfName IEC_TIMER
"IEC_TIMER"
BEGIN
END_DATA_BLOCK

// folder: (top level)

FUNCTION_BLOCK "Blue_PickPlace"   // FB1, LAD
{ S7_Optimized_Access := 'TRUE' }
VERSION : 0.1
   VAR_TEMP   // added for the SCL form of the ladder/FBD networks
      _w1 : Bool;
   END_VAR
BEGIN

REGION Network 1
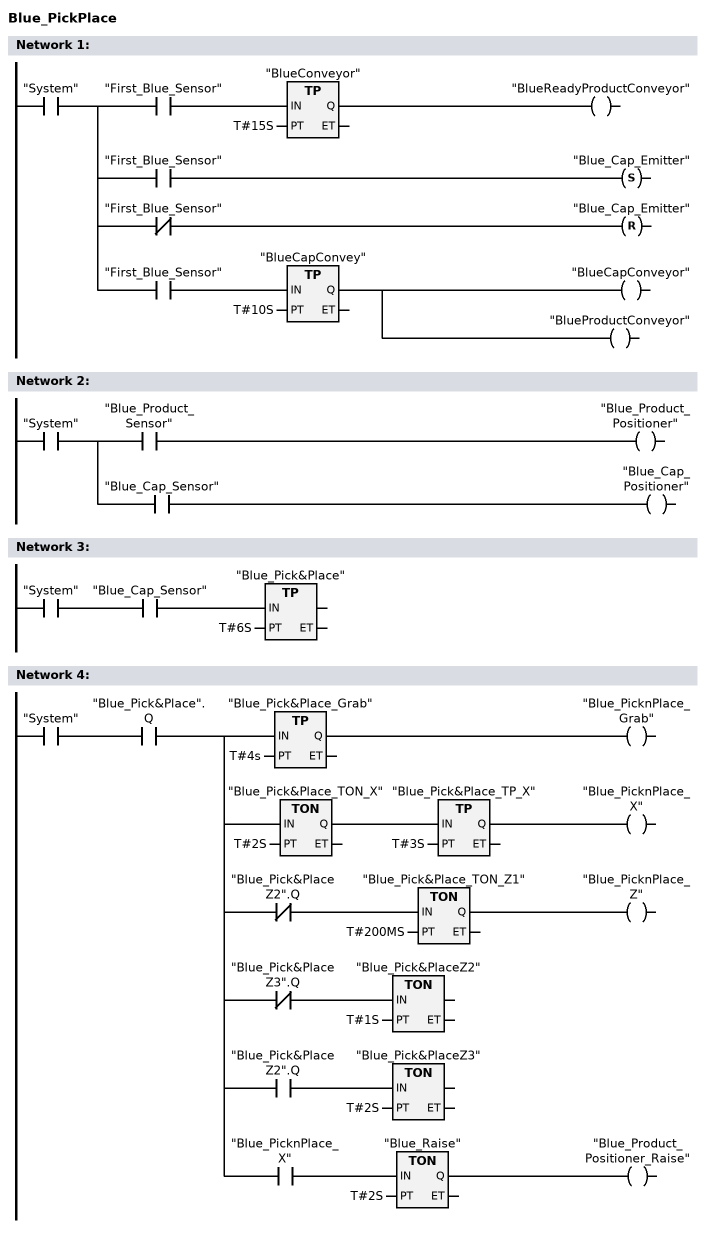
   "BlueConveyor".TP(IN := "System" AND "First_Blue_Sensor", PT := T#15S);
   "BlueReadyProductConveyor" := "BlueConveyor".Q;
   IF "System" AND "First_Blue_Sensor" THEN "Blue_Cap_Emitter" := TRUE; END_IF;
   IF "System" AND NOT "First_Blue_Sensor" THEN "Blue_Cap_Emitter" := FALSE; END_IF;
   "BlueCapConvey".TP(IN := "System" AND "First_Blue_Sensor", PT := T#10S);
   "BlueCapConveyor" := "BlueCapConvey".Q;
   "BlueProductConveyor" := "BlueCapConvey".Q;
END_REGION

REGION Network 2
   RUNG wire#powerrail
      Contact( "System" )
      wire#w1
      Contact( "Blue_Product_Sensor" )
      Coil( "Blue_Product_Positioner" )
   END_RUNG
   RUNG wire#w1
      Contact( "Blue_Cap_Sensor" )
      Coil( "Blue_Cap_Positioner" )
   END_RUNG
   // the same network as SCL:
   "Blue_Product_Positioner" := "System" AND "Blue_Product_Sensor";
   "Blue_Cap_Positioner" := "System" AND "Blue_Cap_Sensor";
END_REGION

REGION Network 3
   "Blue_Pick&Place".TP(IN := "System" AND "Blue_Cap_Sensor", PT := T#6S);
END_REGION

REGION Network 4
   #_w1 := "System" AND "Blue_Pick&Place".Q;
   "Blue_Pick&Place_Grab".TP(IN := #_w1, PT := T#4s);
   "Blue_PicknPlace_Grab" := "Blue_Pick&Place_Grab".Q;
   "Blue_Pick&Place_TON_X".TON(IN := #_w1, PT := T#2S);
   "Blue_Pick&Place_TP_X".TP(IN := "Blue_Pick&Place_TON_X".Q, PT := T#3S);
   "Blue_PicknPlace_X" := "Blue_Pick&Place_TP_X".Q;
   "Blue_Pick&Place_TON_Z1".TON(IN := #_w1 AND NOT "Blue_Pick&PlaceZ2".Q, PT := T#200MS);
   "Blue_PicknPlace_Z" := "Blue_Pick&Place_TON_Z1".Q;
   "Blue_Pick&PlaceZ2".TON(IN := #_w1 AND NOT "Blue_Pick&PlaceZ3".Q, PT := T#1S);
   "Blue_Pick&PlaceZ3".TON(IN := #_w1 AND "Blue_Pick&PlaceZ2".Q, PT := T#2S);
   "Blue_Raise".TON(IN := #_w1 AND "Blue_PicknPlace_X", PT := T#2S);
   "Blue_Product_Positioner_Raise" := "Blue_Raise".Q;
END_REGION
END_FUNCTION_BLOCK

FUNCTION_BLOCK "Blue_Storage_Line"   // FB2, LAD
{ S7_Optimized_Access := 'TRUE' }
VERSION : 0.1
   VAR_TEMP   // added for the SCL form of the ladder/FBD networks
      _w1 : Bool;
   END_VAR
BEGIN

REGION Network 1
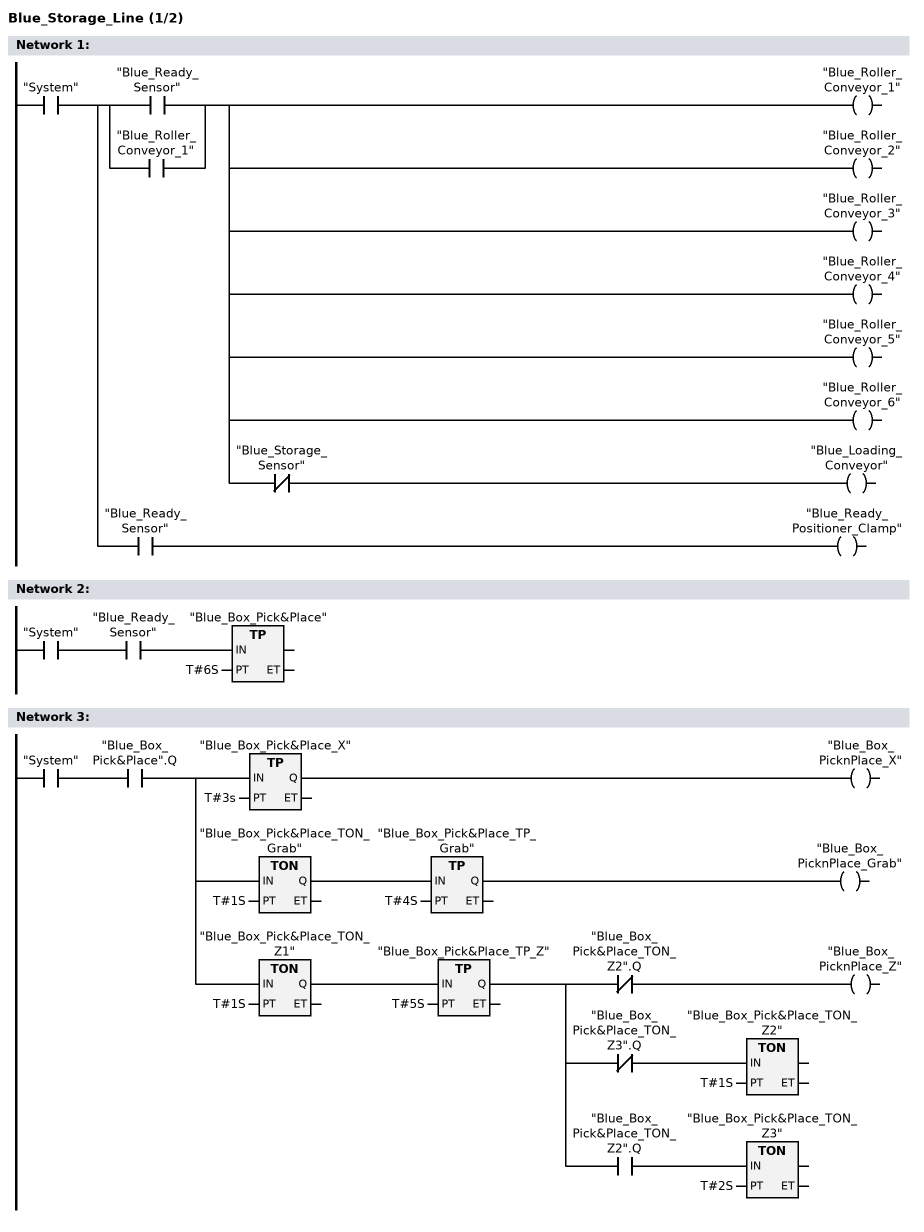
   RUNG wire#powerrail
      Contact( "System" )
      wire#w1
      Contact( "Blue_Ready_Sensor" )
      wire#w2
      Coil( "Blue_Roller_Conveyor_1" )
   END_RUNG
   RUNG wire#w1
      Contact( "Blue_Roller_Conveyor_1" )
   END_RUNG wire#w2
   RUNG wire#w2
      Coil( "Blue_Roller_Conveyor_2" )
   END_RUNG
   RUNG wire#w2
      Coil( "Blue_Roller_Conveyor_3" )
   END_RUNG
   RUNG wire#w2
      Coil( "Blue_Roller_Conveyor_4" )
   END_RUNG
   RUNG wire#w2
      Coil( "Blue_Roller_Conveyor_5" )
   END_RUNG
   RUNG wire#w2
      Coil( "Blue_Roller_Conveyor_6" )
   END_RUNG
   RUNG wire#w2
      I_Contact( "Blue_Storage_Sensor" )
      Coil( "Blue_Loading_Conveyor" )
   END_RUNG
   RUNG wire#w1
      Contact( "Blue_Ready_Sensor" )
      Coil( "Blue_Ready_Positioner_Clamp" )
   END_RUNG
   // the same network as SCL:
   "Blue_Roller_Conveyor_1" := "System" AND ("Blue_Ready_Sensor" OR "Blue_Roller_Conveyor_1");
   "Blue_Roller_Conveyor_2" := "Blue_Roller_Conveyor_1";
   "Blue_Roller_Conveyor_3" := "Blue_Roller_Conveyor_1";
   "Blue_Roller_Conveyor_4" := "Blue_Roller_Conveyor_1";
   "Blue_Roller_Conveyor_5" := "Blue_Roller_Conveyor_1";
   "Blue_Roller_Conveyor_6" := "Blue_Roller_Conveyor_1";
   "Blue_Loading_Conveyor" := "Blue_Roller_Conveyor_1" AND NOT "Blue_Storage_Sensor";
   "Blue_Ready_Positioner_Clamp" := "System" AND "Blue_Ready_Sensor";
END_REGION

REGION Network 2
   "Blue_Box_Pick&Place".TP(IN := "System" AND "Blue_Ready_Sensor", PT := T#6S);
END_REGION

REGION Network 3
   #_w1 := "System" AND "Blue_Box_Pick&Place".Q;
   "Blue_Box_Pick&Place_X".TP(IN := #_w1, PT := T#3s);
   "Blue_Box_PicknPlace_X" := "Blue_Box_Pick&Place_X".Q;
   "Blue_Box_Pick&Place_TON_Grab".TON(IN := #_w1, PT := T#1S);
   "Blue_Box_Pick&Place_TP_Grab".TP(IN := "Blue_Box_Pick&Place_TON_Grab".Q, PT := T#4S);
   "Blue_Box_PicknPlace_Grab" := "Blue_Box_Pick&Place_TP_Grab".Q;
   "Blue_Box_Pick&Place_TON_Z1".TON(IN := #_w1, PT := T#1S);
   "Blue_Box_Pick&Place_TP_Z".TP(IN := "Blue_Box_Pick&Place_TON_Z1".Q, PT := T#5S);
   "Blue_Box_PicknPlace_Z" := "Blue_Box_Pick&Place_TP_Z".Q AND NOT "Blue_Box_Pick&Place_TON_Z2".Q;
   "Blue_Box_Pick&Place_TON_Z2".TON(IN := "Blue_Box_Pick&Place_TP_Z".Q AND NOT "Blue_Box_Pick&Place_TON_Z3".Q,
                           PT := T#1S);
   "Blue_Box_Pick&Place_TON_Z3".TON(IN := "Blue_Box_Pick&Place_TP_Z".Q AND "Blue_Box_Pick&Place_TON_Z2".Q,
                           PT := T#2S);
END_REGION

REGION Network 4
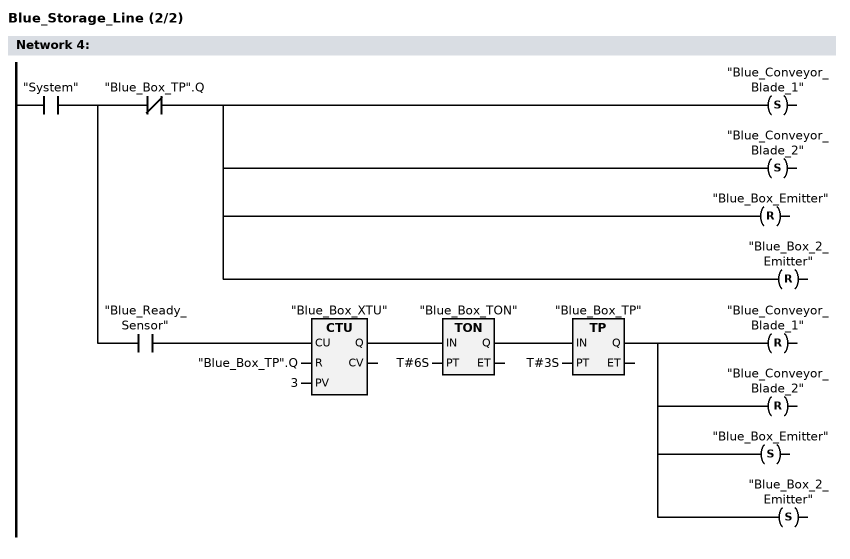
   IF "System" AND NOT "Blue_Box_TP".Q THEN
       "Blue_Conveyor_Blade_1" := TRUE;
       "Blue_Conveyor_Blade_2" := TRUE;
       "Blue_Box_Emitter" := FALSE;
       "Blue_Box_2_Emitter" := FALSE;
   END_IF;
   "Blue_Box_XTU".CTU(CU := "System" AND "Blue_Ready_Sensor", R := "Blue_Box_TP".Q, PV := 3);
   "Blue_Box_TON".TON(IN := "Blue_Box_XTU".Q, PT := T#6S);
   "Blue_Box_TP".TP(IN := "Blue_Box_TON".Q, PT := T#3S);
   IF "Blue_Box_TP".Q THEN
       "Blue_Conveyor_Blade_1" := FALSE;
       "Blue_Conveyor_Blade_2" := FALSE;
       "Blue_Box_Emitter" := TRUE;
       "Blue_Box_2_Emitter" := TRUE;
   END_IF;
END_REGION
END_FUNCTION_BLOCK

FUNCTION_BLOCK "Blue_Store"   // FB3, LAD
{ S7_Optimized_Access := 'TRUE' }
VERSION : 0.1
   VAR_TEMP   // added for the SCL form of the ladder/FBD networks
      _w1 : Bool;
   END_VAR
BEGIN

REGION Network 1
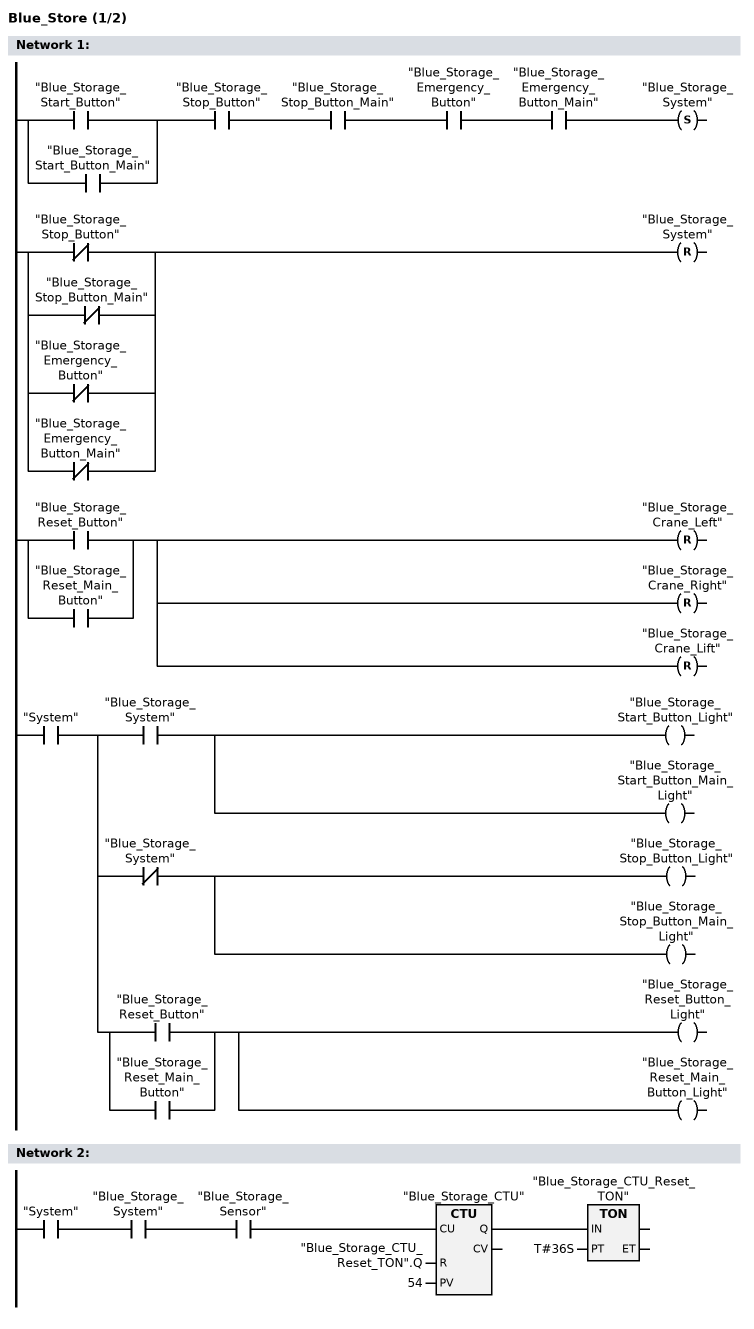
   RUNG wire#powerrail
      Contact( "Blue_Storage_Start_Button" )
      wire#w1
      Contact( "Blue_Storage_Stop_Button" )
      Contact( "Blue_Storage_Stop_Button_Main" )
      Contact( "Blue_Storage_Emergency_Button" )
      Contact( "Blue_Storage_Emergency_Button_Main" )
      S_Coil( "Blue_Storage_System" )
   END_RUNG
   RUNG wire#powerrail
      Contact( "Blue_Storage_Start_Button_Main" )
   END_RUNG wire#w1
   RUNG wire#powerrail
      I_Contact( "Blue_Storage_Stop_Button" )
      wire#w2
      R_Coil( "Blue_Storage_System" )
   END_RUNG
   RUNG wire#powerrail
      I_Contact( "Blue_Storage_Stop_Button_Main" )
   END_RUNG wire#w2
   RUNG wire#powerrail
      I_Contact( "Blue_Storage_Emergency_Button" )
   END_RUNG wire#w2
   RUNG wire#powerrail
      I_Contact( "Blue_Storage_Emergency_Button_Main" )
   END_RUNG wire#w2
   RUNG wire#powerrail
      Contact( "Blue_Storage_Reset_Button" )
      wire#w3
      R_Coil( "Blue_Storage_Crane_Left" )
   END_RUNG
   RUNG wire#powerrail
      Contact( "Blue_Storage_Reset_Main_Button" )
   END_RUNG wire#w3
   RUNG wire#w3
      R_Coil( "Blue_Storage_Crane_Right" )
   END_RUNG
   RUNG wire#w3
      R_Coil( "Blue_Storage_Crane_Lift" )
   END_RUNG
   RUNG wire#powerrail
      Contact( "System" )
      wire#w4
      Contact( "Blue_Storage_System" )
      wire#w5
      Coil( "Blue_Storage_Start_Button_Light" )
   END_RUNG
   RUNG wire#w5
      Coil( "Blue_Storage_Start_Button_Main_Light" )
   END_RUNG
   RUNG wire#w4
      I_Contact( "Blue_Storage_System" )
      wire#w6
      Coil( "Blue_Storage_Stop_Button_Light" )
   END_RUNG
   RUNG wire#w6
      Coil( "Blue_Storage_Stop_Button_Main_Light" )
   END_RUNG
   RUNG wire#w4
      Contact( "Blue_Storage_Reset_Button" )
      wire#w7
      Coil( "Blue_Storage_Reset_Button_Light" )
   END_RUNG
   RUNG wire#w4
      Contact( "Blue_Storage_Reset_Main_Button" )
   END_RUNG wire#w7
   RUNG wire#w7
      Coil( "Blue_Storage_Reset_Main_Button_Light" )
   END_RUNG
   // the same network as SCL:
   IF ("Blue_Storage_Start_Button" OR "Blue_Storage_Start_Button_Main") AND "Blue_Storage_Stop_Button" AND "Blue_Storage_Stop_Button_Main" AND "Blue_Storage_Emergency_Button" AND "Blue_Storage_Emergency_Button_Main" THEN
       "Blue_Storage_System" := TRUE;
   END_IF;
   IF NOT "Blue_Storage_Stop_Button" OR NOT "Blue_Storage_Stop_Button_Main" OR NOT "Blue_Storage_Emergency_Button" OR NOT "Blue_Storage_Emergency_Button_Main" THEN
       "Blue_Storage_System" := FALSE;
   END_IF;
   IF "Blue_Storage_Reset_Button" OR "Blue_Storage_Reset_Main_Button" THEN
       "Blue_Storage_Crane_Left" := FALSE;
       "Blue_Storage_Crane_Right" := FALSE;
       "Blue_Storage_Crane_Lift" := FALSE;
   END_IF;
   "Blue_Storage_Start_Button_Light" := "System" AND "Blue_Storage_System";
   "Blue_Storage_Start_Button_Main_Light" := "Blue_Storage_Start_Button_Light";
   "Blue_Storage_Stop_Button_Light" := "System" AND NOT "Blue_Storage_System";
   "Blue_Storage_Stop_Button_Main_Light" := "Blue_Storage_Stop_Button_Light";
   "Blue_Storage_Reset_Button_Light" := "System" AND ("Blue_Storage_Reset_Button" OR "Blue_Storage_Reset_Main_Button");
   "Blue_Storage_Reset_Main_Button_Light" := "Blue_Storage_Reset_Button_Light";
END_REGION

REGION Network 2
   "Blue_Storage_CTU".CTU(CU := "System" AND "Blue_Storage_System" AND "Blue_Storage_Sensor",
                          R := "Blue_Storage_CTU_Reset_TON".Q,
                          PV := 54);
   "Blue_Storage_CTU_Reset_TON".TON(IN := "Blue_Storage_CTU".Q, PT := T#36S);
END_REGION

REGION Network 3
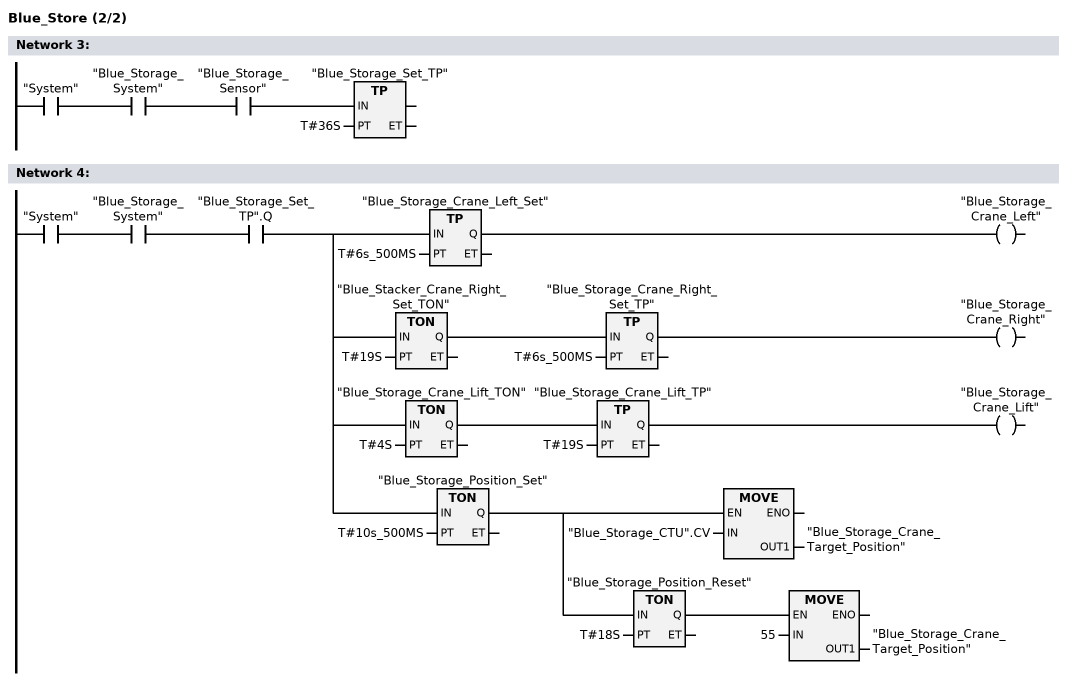
   "Blue_Storage_Set_TP".TP(IN := "System" AND "Blue_Storage_System" AND "Blue_Storage_Sensor", PT := T#36S);
END_REGION

REGION Network 4
   #_w1 := "System" AND "Blue_Storage_System" AND "Blue_Storage_Set_TP".Q;
   "Blue_Storage_Crane_Left_Set".TP(IN := #_w1, PT := T#6s_500MS);
   "Blue_Storage_Crane_Left" := "Blue_Storage_Crane_Left_Set".Q;
   "Blue_Stacker_Crane_Right_Set_TON".TON(IN := #_w1, PT := T#19S);
   "Blue_Storage_Crane_Right_Set_TP".TP(IN := "Blue_Stacker_Crane_Right_Set_TON".Q, PT := T#6s_500MS);
   "Blue_Storage_Crane_Right" := "Blue_Storage_Crane_Right_Set_TP".Q;
   "Blue_Storage_Crane_Lift_TON".TON(IN := #_w1, PT := T#4S);
   "Blue_Storage_Crane_Lift_TP".TP(IN := "Blue_Storage_Crane_Lift_TON".Q, PT := T#19S);
   "Blue_Storage_Crane_Lift" := "Blue_Storage_Crane_Lift_TP".Q;
   "Blue_Storage_Position_Set".TON(IN := #_w1, PT := T#10s_500MS);
   IF "Blue_Storage_Position_Set".Q THEN
       "Blue_Storage_Crane_Target_Position" := "Blue_Storage_CTU".CV;
   END_IF;
   "Blue_Storage_Position_Reset".TON(IN := "Blue_Storage_Position_Set".Q, PT := T#18S);
   IF "Blue_Storage_Position_Reset".Q THEN "Blue_Storage_Crane_Target_Position" := 55; END_IF;
END_REGION
END_FUNCTION_BLOCK

FUNCTION_BLOCK "Gray_PickPlace"   // FB4, LAD
{ S7_Optimized_Access := 'TRUE' }
VERSION : 0.1
   VAR_TEMP   // added for the SCL form of the ladder/FBD networks
      _w1 : Bool;
   END_VAR
BEGIN

REGION Network 1
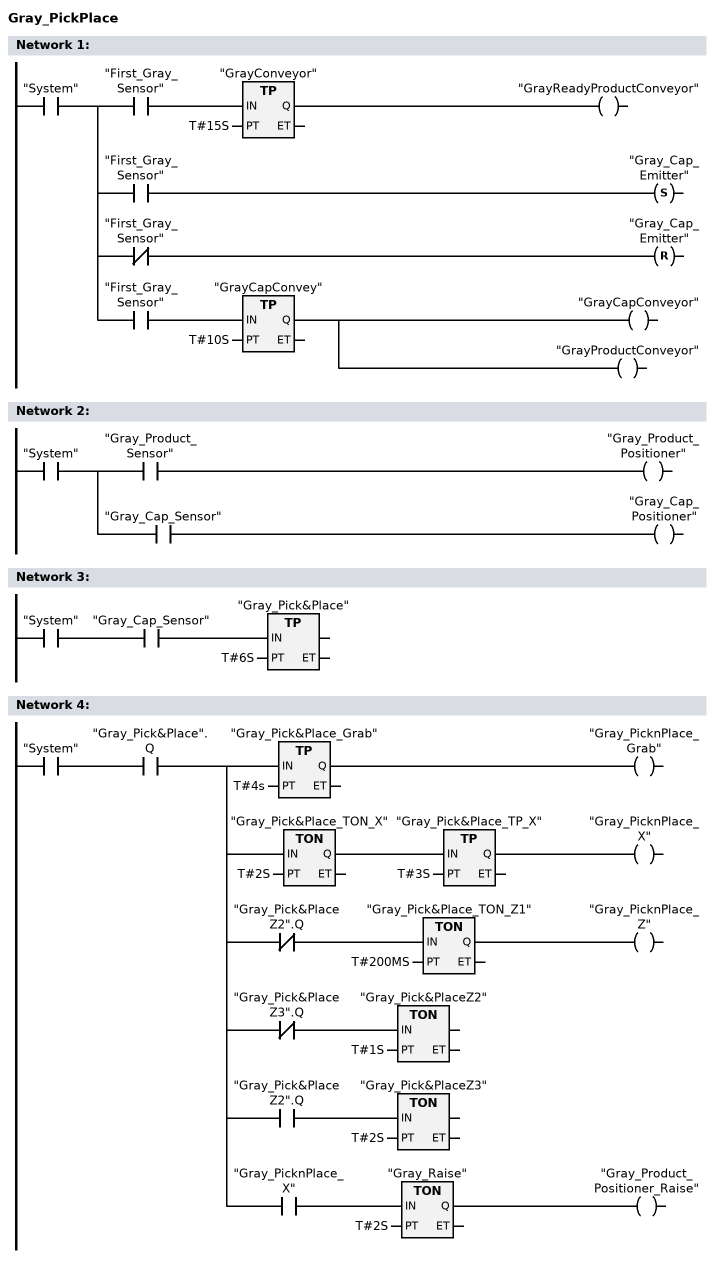
   "GrayConveyor".TP(IN := "System" AND "First_Gray_Sensor", PT := T#15S);
   "GrayReadyProductConveyor" := "GrayConveyor".Q;
   IF "System" AND "First_Gray_Sensor" THEN "Gray_Cap_Emitter" := TRUE; END_IF;
   IF "System" AND NOT "First_Gray_Sensor" THEN "Gray_Cap_Emitter" := FALSE; END_IF;
   "GrayCapConvey".TP(IN := "System" AND "First_Gray_Sensor", PT := T#10S);
   "GrayCapConveyor" := "GrayCapConvey".Q;
   "GrayProductConveyor" := "GrayCapConvey".Q;
END_REGION

REGION Network 2
   RUNG wire#powerrail
      Contact( "System" )
      wire#w1
      Contact( "Gray_Product_Sensor" )
      Coil( "Gray_Product_Positioner" )
   END_RUNG
   RUNG wire#w1
      Contact( "Gray_Cap_Sensor" )
      Coil( "Gray_Cap_Positioner" )
   END_RUNG
   // the same network as SCL:
   "Gray_Product_Positioner" := "System" AND "Gray_Product_Sensor";
   "Gray_Cap_Positioner" := "System" AND "Gray_Cap_Sensor";
END_REGION

REGION Network 3
   "Gray_Pick&Place".TP(IN := "System" AND "Gray_Cap_Sensor", PT := T#6S);
END_REGION

REGION Network 4
   #_w1 := "System" AND "Gray_Pick&Place".Q;
   "Gray_Pick&Place_Grab".TP(IN := #_w1, PT := T#4s);
   "Gray_PicknPlace_Grab" := "Gray_Pick&Place_Grab".Q;
   "Gray_Pick&Place_TON_X".TON(IN := #_w1, PT := T#2S);
   "Gray_Pick&Place_TP_X".TP(IN := "Gray_Pick&Place_TON_X".Q, PT := T#3S);
   "Gray_PicknPlace_X" := "Gray_Pick&Place_TP_X".Q;
   "Gray_Pick&Place_TON_Z1".TON(IN := #_w1 AND NOT "Gray_Pick&PlaceZ2".Q, PT := T#200MS);
   "Gray_PicknPlace_Z" := "Gray_Pick&Place_TON_Z1".Q;
   "Gray_Pick&PlaceZ2".TON(IN := #_w1 AND NOT "Gray_Pick&PlaceZ3".Q, PT := T#1S);
   "Gray_Pick&PlaceZ3".TON(IN := #_w1 AND "Gray_Pick&PlaceZ2".Q, PT := T#2S);
   "Gray_Raise".TON(IN := #_w1 AND "Gray_PicknPlace_X", PT := T#2S);
   "Gray_Product_Positioner_Raise" := "Gray_Raise".Q;
END_REGION
END_FUNCTION_BLOCK

FUNCTION_BLOCK "Gray_Storage_Line"   // FB5, LAD
{ S7_Optimized_Access := 'TRUE' }
VERSION : 0.1
   VAR_TEMP   // added for the SCL form of the ladder/FBD networks
      _w1 : Bool;
   END_VAR
BEGIN

REGION Network 1
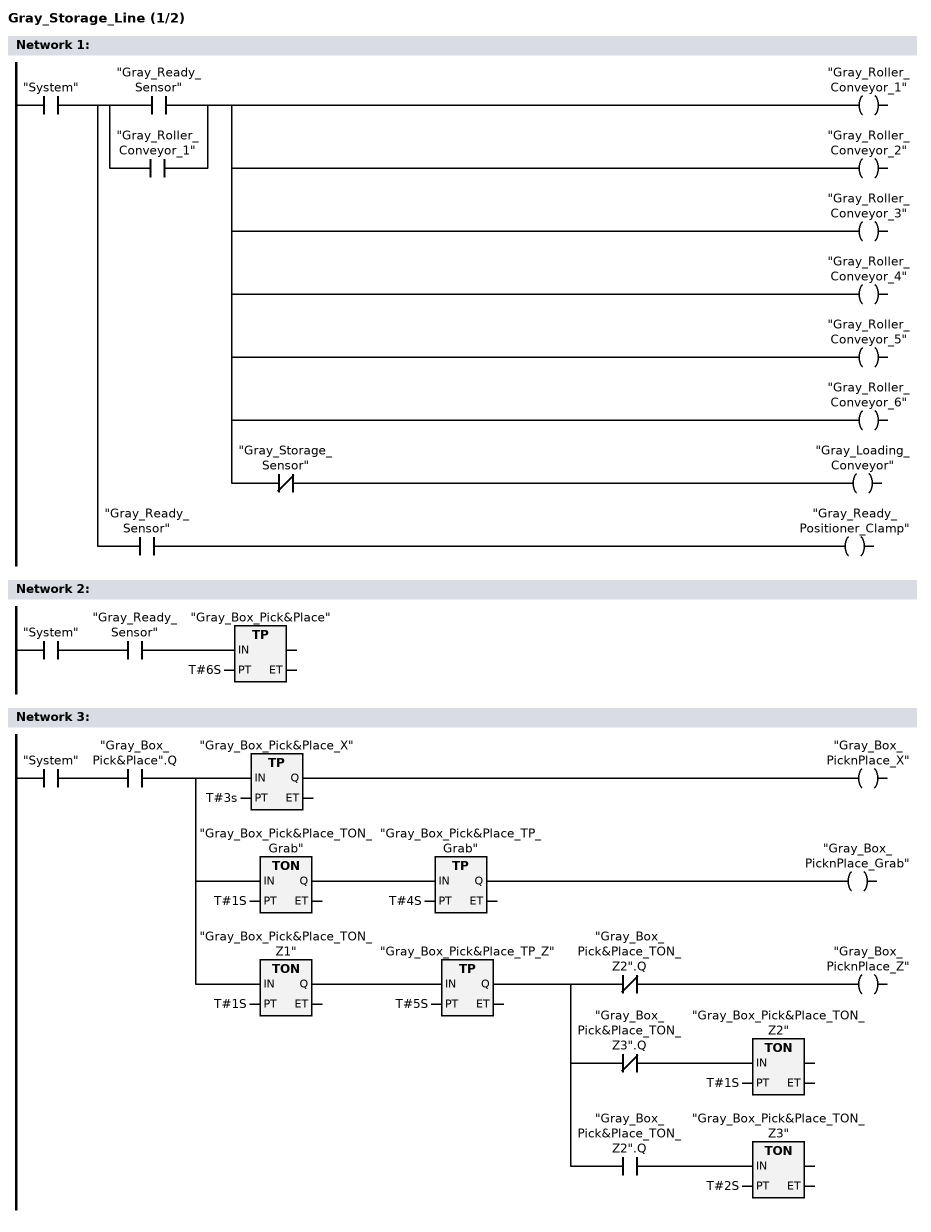
   RUNG wire#powerrail
      Contact( "System" )
      wire#w1
      Contact( "Gray_Ready_Sensor" )
      wire#w2
      Coil( "Gray_Roller_Conveyor_1" )
   END_RUNG
   RUNG wire#w1
      Contact( "Gray_Roller_Conveyor_1" )
   END_RUNG wire#w2
   RUNG wire#w2
      Coil( "Gray_Roller_Conveyor_2" )
   END_RUNG
   RUNG wire#w2
      Coil( "Gray_Roller_Conveyor_3" )
   END_RUNG
   RUNG wire#w2
      Coil( "Gray_Roller_Conveyor_4" )
   END_RUNG
   RUNG wire#w2
      Coil( "Gray_Roller_Conveyor_5" )
   END_RUNG
   RUNG wire#w2
      Coil( "Gray_Roller_Conveyor_6" )
   END_RUNG
   RUNG wire#w2
      I_Contact( "Gray_Storage_Sensor" )
      Coil( "Gray_Loading_Conveyor" )
   END_RUNG
   RUNG wire#w1
      Contact( "Gray_Ready_Sensor" )
      Coil( "Gray_Ready_Positioner_Clamp" )
   END_RUNG
   // the same network as SCL:
   "Gray_Roller_Conveyor_1" := "System" AND ("Gray_Ready_Sensor" OR "Gray_Roller_Conveyor_1");
   "Gray_Roller_Conveyor_2" := "Gray_Roller_Conveyor_1";
   "Gray_Roller_Conveyor_3" := "Gray_Roller_Conveyor_1";
   "Gray_Roller_Conveyor_4" := "Gray_Roller_Conveyor_1";
   "Gray_Roller_Conveyor_5" := "Gray_Roller_Conveyor_1";
   "Gray_Roller_Conveyor_6" := "Gray_Roller_Conveyor_1";
   "Gray_Loading_Conveyor" := "Gray_Roller_Conveyor_1" AND NOT "Gray_Storage_Sensor";
   "Gray_Ready_Positioner_Clamp" := "System" AND "Gray_Ready_Sensor";
END_REGION

REGION Network 2
   "Gray_Box_Pick&Place".TP(IN := "System" AND "Gray_Ready_Sensor", PT := T#6S);
END_REGION

REGION Network 3
   #_w1 := "System" AND "Gray_Box_Pick&Place".Q;
   "Gray_Box_Pick&Place_X".TP(IN := #_w1, PT := T#3s);
   "Gray_Box_PicknPlace_X" := "Gray_Box_Pick&Place_X".Q;
   "Gray_Box_Pick&Place_TON_Grab".TON(IN := #_w1, PT := T#1S);
   "Gray_Box_Pick&Place_TP_Grab".TP(IN := "Gray_Box_Pick&Place_TON_Grab".Q, PT := T#4S);
   "Gray_Box_PicknPlace_Grab" := "Gray_Box_Pick&Place_TP_Grab".Q;
   "Gray_Box_Pick&Place_TON_Z1".TON(IN := #_w1, PT := T#1S);
   "Gray_Box_Pick&Place_TP_Z".TP(IN := "Gray_Box_Pick&Place_TON_Z1".Q, PT := T#5S);
   "Gray_Box_PicknPlace_Z" := "Gray_Box_Pick&Place_TP_Z".Q AND NOT "Gray_Box_Pick&Place_TON_Z2".Q;
   "Gray_Box_Pick&Place_TON_Z2".TON(IN := "Gray_Box_Pick&Place_TP_Z".Q AND NOT "Gray_Box_Pick&Place_TON_Z3".Q,
                           PT := T#1S);
   "Gray_Box_Pick&Place_TON_Z3".TON(IN := "Gray_Box_Pick&Place_TP_Z".Q AND "Gray_Box_Pick&Place_TON_Z2".Q,
                           PT := T#2S);
END_REGION

REGION Network 4
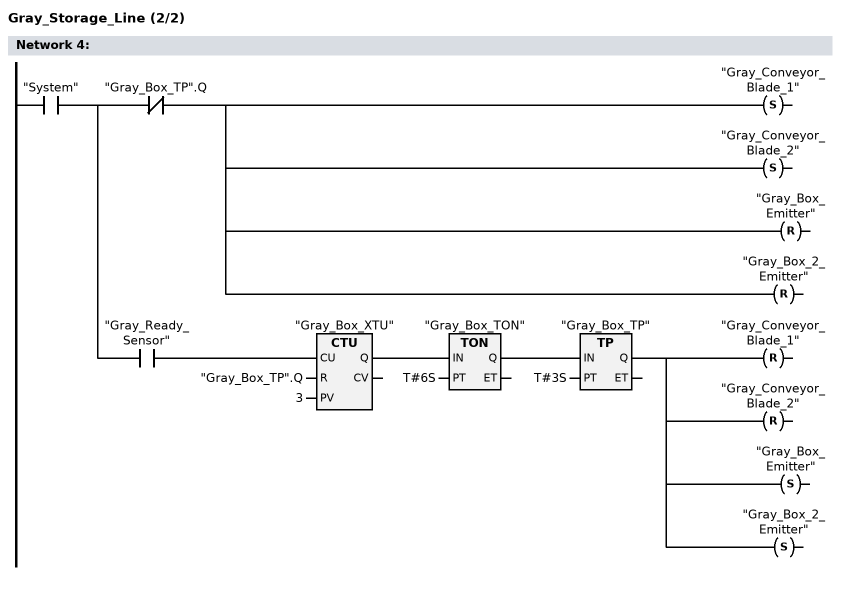
   IF "System" AND NOT "Gray_Box_TP".Q THEN
       "Gray_Conveyor_Blade_1" := TRUE;
       "Gray_Conveyor_Blade_2" := TRUE;
       "Gray_Box_Emitter" := FALSE;
       "Gray_Box_2_Emitter" := FALSE;
   END_IF;
   "Gray_Box_XTU".CTU(CU := "System" AND "Gray_Ready_Sensor", R := "Gray_Box_TP".Q, PV := 3);
   "Gray_Box_TON".TON(IN := "Gray_Box_XTU".Q, PT := T#6S);
   "Gray_Box_TP".TP(IN := "Gray_Box_TON".Q, PT := T#3S);
   IF "Gray_Box_TP".Q THEN
       "Gray_Conveyor_Blade_1" := FALSE;
       "Gray_Conveyor_Blade_2" := FALSE;
       "Gray_Box_Emitter" := TRUE;
       "Gray_Box_2_Emitter" := TRUE;
   END_IF;
END_REGION
END_FUNCTION_BLOCK

FUNCTION_BLOCK "Gray_Store"   // FB6, LAD
{ S7_Optimized_Access := 'TRUE' }
VERSION : 0.1
   VAR_TEMP   // added for the SCL form of the ladder/FBD networks
      _w1 : Bool;
   END_VAR
BEGIN

REGION Network 1
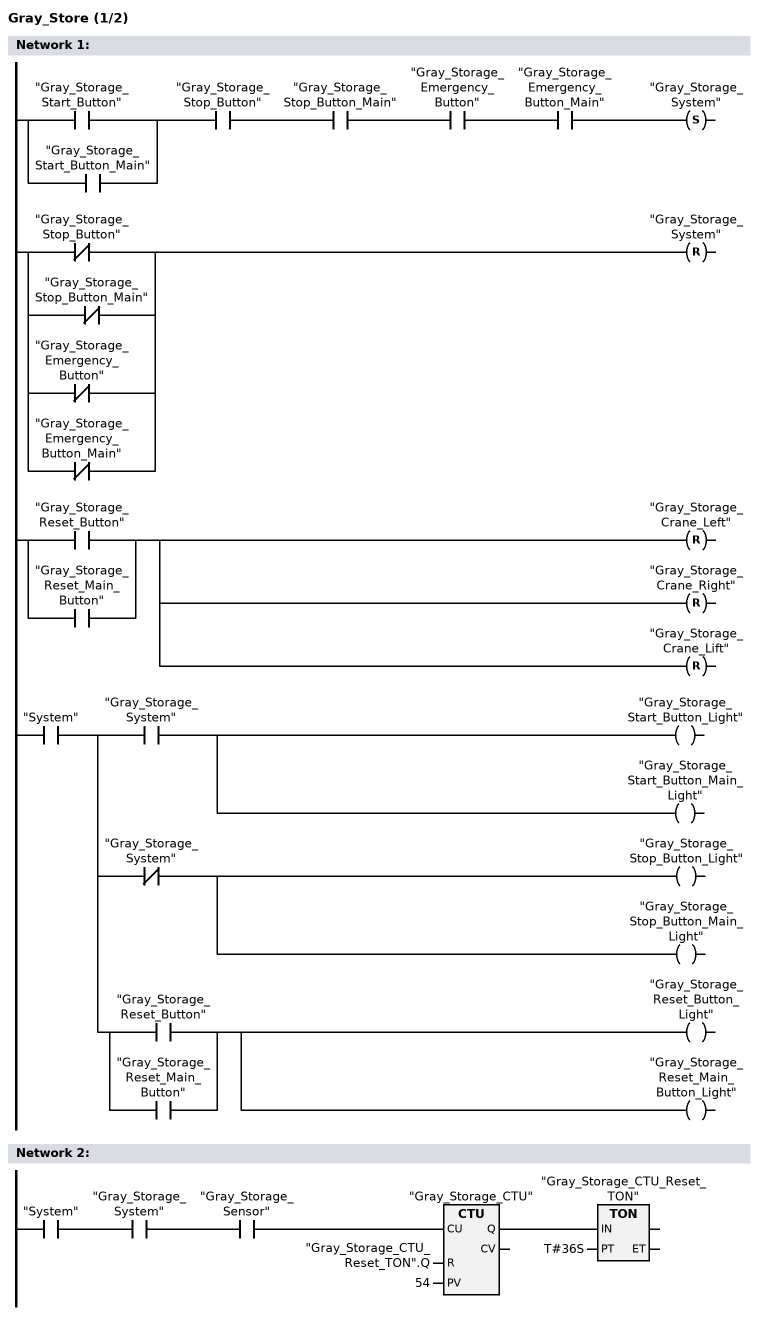
   RUNG wire#powerrail
      Contact( "Gray_Storage_Start_Button" )
      wire#w1
      Contact( "Gray_Storage_Stop_Button" )
      Contact( "Gray_Storage_Stop_Button_Main" )
      Contact( "Gray_Storage_Emergency_Button" )
      Contact( "Gray_Storage_Emergency_Button_Main" )
      S_Coil( "Gray_Storage_System" )
   END_RUNG
   RUNG wire#powerrail
      Contact( "Gray_Storage_Start_Button_Main" )
   END_RUNG wire#w1
   RUNG wire#powerrail
      I_Contact( "Gray_Storage_Stop_Button" )
      wire#w2
      R_Coil( "Gray_Storage_System" )
   END_RUNG
   RUNG wire#powerrail
      I_Contact( "Gray_Storage_Stop_Button_Main" )
   END_RUNG wire#w2
   RUNG wire#powerrail
      I_Contact( "Gray_Storage_Emergency_Button" )
   END_RUNG wire#w2
   RUNG wire#powerrail
      I_Contact( "Gray_Storage_Emergency_Button_Main" )
   END_RUNG wire#w2
   RUNG wire#powerrail
      Contact( "Gray_Storage_Reset_Button" )
      wire#w3
      R_Coil( "Gray_Storage_Crane_Left" )
   END_RUNG
   RUNG wire#powerrail
      Contact( "Gray_Storage_Reset_Main_Button" )
   END_RUNG wire#w3
   RUNG wire#w3
      R_Coil( "Gray_Storage_Crane_Right" )
   END_RUNG
   RUNG wire#w3
      R_Coil( "Gray_Storage_Crane_Lift" )
   END_RUNG
   RUNG wire#powerrail
      Contact( "System" )
      wire#w4
      Contact( "Gray_Storage_System" )
      wire#w5
      Coil( "Gray_Storage_Start_Button_Light" )
   END_RUNG
   RUNG wire#w5
      Coil( "Gray_Storage_Start_Button_Main_Light" )
   END_RUNG
   RUNG wire#w4
      I_Contact( "Gray_Storage_System" )
      wire#w6
      Coil( "Gray_Storage_Stop_Button_Light" )
   END_RUNG
   RUNG wire#w6
      Coil( "Gray_Storage_Stop_Button_Main_Light" )
   END_RUNG
   RUNG wire#w4
      Contact( "Gray_Storage_Reset_Button" )
      wire#w7
      Coil( "Gray_Storage_Reset_Button_Light" )
   END_RUNG
   RUNG wire#w4
      Contact( "Gray_Storage_Reset_Main_Button" )
   END_RUNG wire#w7
   RUNG wire#w7
      Coil( "Gray_Storage_Reset_Main_Button_Light" )
   END_RUNG
   // the same network as SCL:
   IF ("Gray_Storage_Start_Button" OR "Gray_Storage_Start_Button_Main") AND "Gray_Storage_Stop_Button" AND "Gray_Storage_Stop_Button_Main" AND "Gray_Storage_Emergency_Button" AND "Gray_Storage_Emergency_Button_Main" THEN
       "Gray_Storage_System" := TRUE;
   END_IF;
   IF NOT "Gray_Storage_Stop_Button" OR NOT "Gray_Storage_Stop_Button_Main" OR NOT "Gray_Storage_Emergency_Button" OR NOT "Gray_Storage_Emergency_Button_Main" THEN
       "Gray_Storage_System" := FALSE;
   END_IF;
   IF "Gray_Storage_Reset_Button" OR "Gray_Storage_Reset_Main_Button" THEN
       "Gray_Storage_Crane_Left" := FALSE;
       "Gray_Storage_Crane_Right" := FALSE;
       "Gray_Storage_Crane_Lift" := FALSE;
   END_IF;
   "Gray_Storage_Start_Button_Light" := "System" AND "Gray_Storage_System";
   "Gray_Storage_Start_Button_Main_Light" := "Gray_Storage_Start_Button_Light";
   "Gray_Storage_Stop_Button_Light" := "System" AND NOT "Gray_Storage_System";
   "Gray_Storage_Stop_Button_Main_Light" := "Gray_Storage_Stop_Button_Light";
   "Gray_Storage_Reset_Button_Light" := "System" AND ("Gray_Storage_Reset_Button" OR "Gray_Storage_Reset_Main_Button");
   "Gray_Storage_Reset_Main_Button_Light" := "Gray_Storage_Reset_Button_Light";
END_REGION

REGION Network 2
   "Gray_Storage_CTU".CTU(CU := "System" AND "Gray_Storage_System" AND "Gray_Storage_Sensor",
                          R := "Gray_Storage_CTU_Reset_TON".Q,
                          PV := 54);
   "Gray_Storage_CTU_Reset_TON".TON(IN := "Gray_Storage_CTU".Q, PT := T#36S);
END_REGION

REGION Network 3
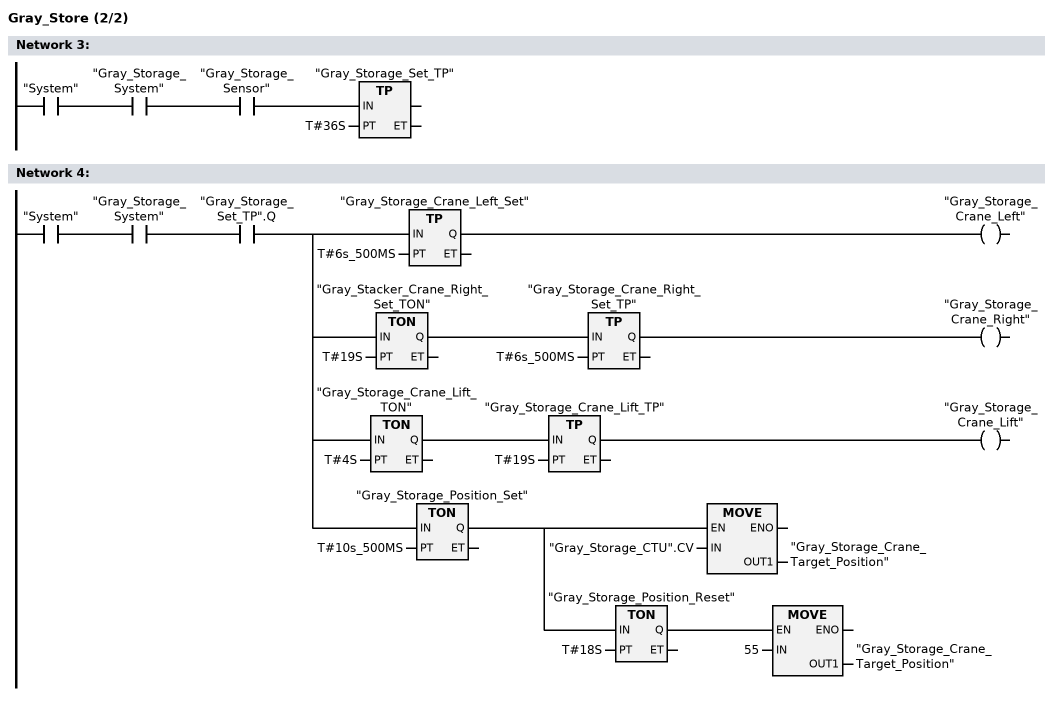
   "Gray_Storage_Set_TP".TP(IN := "System" AND "Gray_Storage_System" AND "Gray_Storage_Sensor", PT := T#36S);
END_REGION

REGION Network 4
   #_w1 := "System" AND "Gray_Storage_System" AND "Gray_Storage_Set_TP".Q;
   "Gray_Storage_Crane_Left_Set".TP(IN := #_w1, PT := T#6s_500MS);
   "Gray_Storage_Crane_Left" := "Gray_Storage_Crane_Left_Set".Q;
   "Gray_Stacker_Crane_Right_Set_TON".TON(IN := #_w1, PT := T#19S);
   "Gray_Storage_Crane_Right_Set_TP".TP(IN := "Gray_Stacker_Crane_Right_Set_TON".Q, PT := T#6s_500MS);
   "Gray_Storage_Crane_Right" := "Gray_Storage_Crane_Right_Set_TP".Q;
   "Gray_Storage_Crane_Lift_TON".TON(IN := #_w1, PT := T#4S);
   "Gray_Storage_Crane_Lift_TP".TP(IN := "Gray_Storage_Crane_Lift_TON".Q, PT := T#19S);
   "Gray_Storage_Crane_Lift" := "Gray_Storage_Crane_Lift_TP".Q;
   "Gray_Storage_Position_Set".TON(IN := #_w1, PT := T#10s_500MS);
   IF "Gray_Storage_Position_Set".Q THEN
       "Gray_Storage_Crane_Target_Position" := "Gray_Storage_CTU".CV;
   END_IF;
   "Gray_Storage_Position_Reset".TON(IN := "Gray_Storage_Position_Set".Q, PT := T#18S);
   IF "Gray_Storage_Position_Reset".Q THEN "Gray_Storage_Crane_Target_Position" := 55; END_IF;
END_REGION
END_FUNCTION_BLOCK

FUNCTION_BLOCK "Green_PickPlace"   // FB7, LAD
{ S7_Optimized_Access := 'TRUE' }
VERSION : 0.1
   VAR_TEMP   // added for the SCL form of the ladder/FBD networks
      _w1 : Bool;
   END_VAR
BEGIN

REGION Network 1
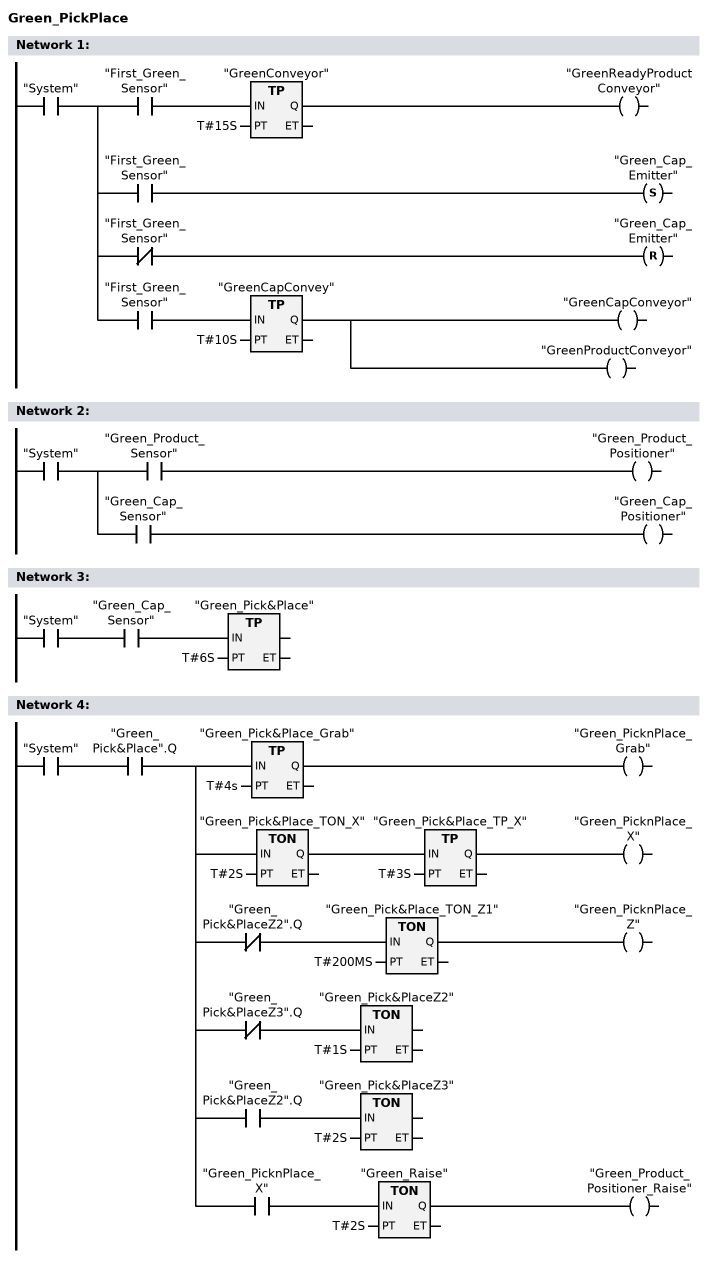
   "GreenConveyor".TP(IN := "System" AND "First_Green_Sensor", PT := T#15S);
   "GreenReadyProductConveyor" := "GreenConveyor".Q;
   IF "System" AND "First_Green_Sensor" THEN "Green_Cap_Emitter" := TRUE; END_IF;
   IF "System" AND NOT "First_Green_Sensor" THEN "Green_Cap_Emitter" := FALSE; END_IF;
   "GreenCapConvey".TP(IN := "System" AND "First_Green_Sensor", PT := T#10S);
   "GreenCapConveyor" := "GreenCapConvey".Q;
   "GreenProductConveyor" := "GreenCapConvey".Q;
END_REGION

REGION Network 2
   RUNG wire#powerrail
      Contact( "System" )
      wire#w1
      Contact( "Green_Product_Sensor" )
      Coil( "Green_Product_Positioner" )
   END_RUNG
   RUNG wire#w1
      Contact( "Green_Cap_Sensor" )
      Coil( "Green_Cap_Positioner" )
   END_RUNG
   // the same network as SCL:
   "Green_Product_Positioner" := "System" AND "Green_Product_Sensor";
   "Green_Cap_Positioner" := "System" AND "Green_Cap_Sensor";
END_REGION

REGION Network 3
   "Green_Pick&Place".TP(IN := "System" AND "Green_Cap_Sensor", PT := T#6S);
END_REGION

REGION Network 4
   #_w1 := "System" AND "Green_Pick&Place".Q;
   "Green_Pick&Place_Grab".TP(IN := #_w1, PT := T#4s);
   "Green_PicknPlace_Grab" := "Green_Pick&Place_Grab".Q;
   "Green_Pick&Place_TON_X".TON(IN := #_w1, PT := T#2S);
   "Green_Pick&Place_TP_X".TP(IN := "Green_Pick&Place_TON_X".Q, PT := T#3S);
   "Green_PicknPlace_X" := "Green_Pick&Place_TP_X".Q;
   "Green_Pick&Place_TON_Z1".TON(IN := #_w1 AND NOT "Green_Pick&PlaceZ2".Q, PT := T#200MS);
   "Green_PicknPlace_Z" := "Green_Pick&Place_TON_Z1".Q;
   "Green_Pick&PlaceZ2".TON(IN := #_w1 AND NOT "Green_Pick&PlaceZ3".Q, PT := T#1S);
   "Green_Pick&PlaceZ3".TON(IN := #_w1 AND "Green_Pick&PlaceZ2".Q, PT := T#2S);
   "Green_Raise".TON(IN := #_w1 AND "Green_PicknPlace_X", PT := T#2S);
   "Green_Product_Positioner_Raise" := "Green_Raise".Q;
END_REGION
END_FUNCTION_BLOCK

FUNCTION_BLOCK "Green_Storage_Line"   // FB8, LAD
{ S7_Optimized_Access := 'TRUE' }
VERSION : 0.1
   VAR_TEMP   // added for the SCL form of the ladder/FBD networks
      _w1 : Bool;
   END_VAR
BEGIN

REGION Network 1
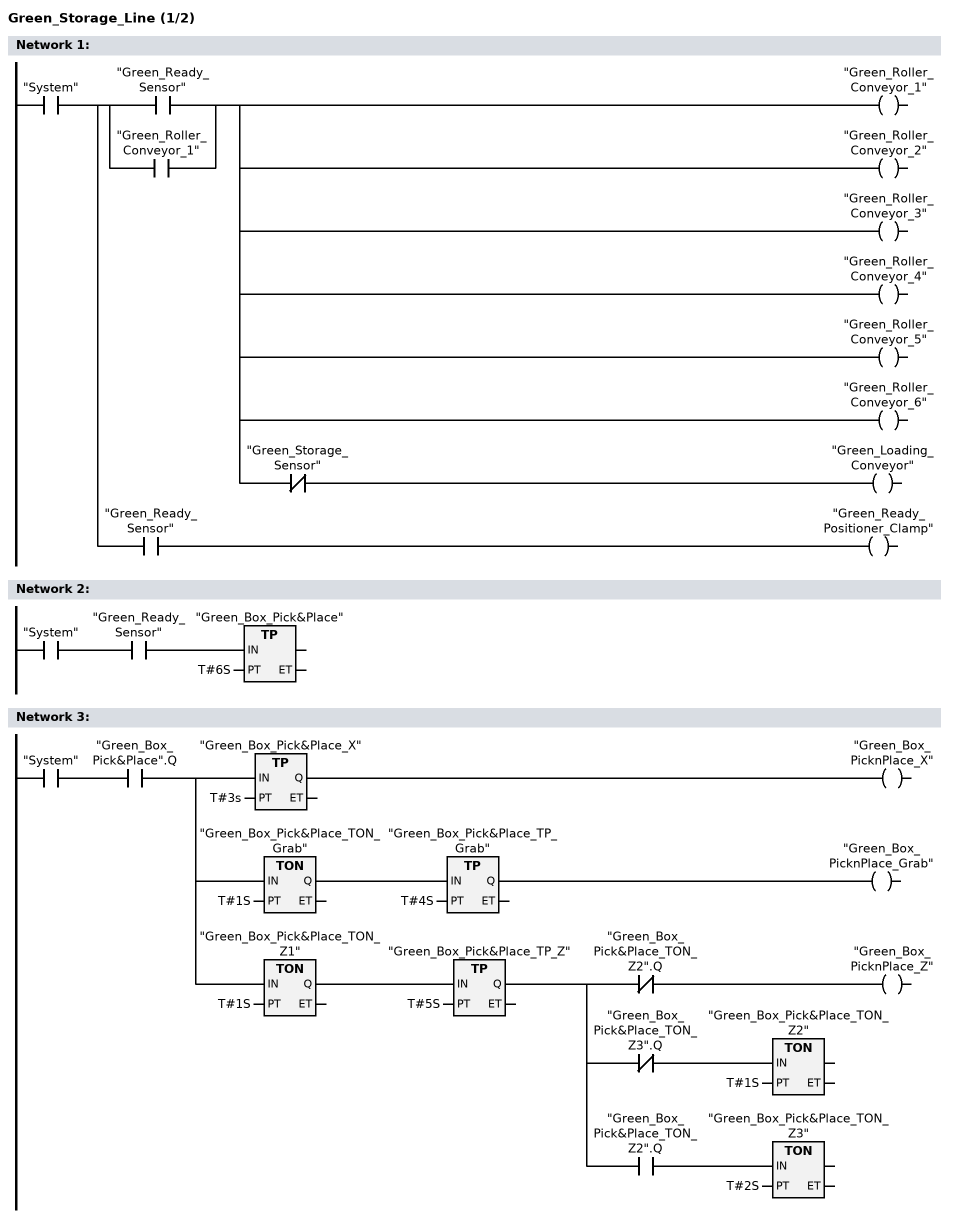
   RUNG wire#powerrail
      Contact( "System" )
      wire#w1
      Contact( "Green_Ready_Sensor" )
      wire#w2
      Coil( "Green_Roller_Conveyor_1" )
   END_RUNG
   RUNG wire#w1
      Contact( "Green_Roller_Conveyor_1" )
   END_RUNG wire#w2
   RUNG wire#w2
      Coil( "Green_Roller_Conveyor_2" )
   END_RUNG
   RUNG wire#w2
      Coil( "Green_Roller_Conveyor_3" )
   END_RUNG
   RUNG wire#w2
      Coil( "Green_Roller_Conveyor_4" )
   END_RUNG
   RUNG wire#w2
      Coil( "Green_Roller_Conveyor_5" )
   END_RUNG
   RUNG wire#w2
      Coil( "Green_Roller_Conveyor_6" )
   END_RUNG
   RUNG wire#w2
      I_Contact( "Green_Storage_Sensor" )
      Coil( "Green_Loading_Conveyor" )
   END_RUNG
   RUNG wire#w1
      Contact( "Green_Ready_Sensor" )
      Coil( "Green_Ready_Positioner_Clamp" )
   END_RUNG
   // the same network as SCL:
   "Green_Roller_Conveyor_1" := "System" AND ("Green_Ready_Sensor" OR "Green_Roller_Conveyor_1");
   "Green_Roller_Conveyor_2" := "Green_Roller_Conveyor_1";
   "Green_Roller_Conveyor_3" := "Green_Roller_Conveyor_1";
   "Green_Roller_Conveyor_4" := "Green_Roller_Conveyor_1";
   "Green_Roller_Conveyor_5" := "Green_Roller_Conveyor_1";
   "Green_Roller_Conveyor_6" := "Green_Roller_Conveyor_1";
   "Green_Loading_Conveyor" := "Green_Roller_Conveyor_1" AND NOT "Green_Storage_Sensor";
   "Green_Ready_Positioner_Clamp" := "System" AND "Green_Ready_Sensor";
END_REGION

REGION Network 2
   "Green_Box_Pick&Place".TP(IN := "System" AND "Green_Ready_Sensor", PT := T#6S);
END_REGION

REGION Network 3
   #_w1 := "System" AND "Green_Box_Pick&Place".Q;
   "Green_Box_Pick&Place_X".TP(IN := #_w1, PT := T#3s);
   "Green_Box_PicknPlace_X" := "Green_Box_Pick&Place_X".Q;
   "Green_Box_Pick&Place_TON_Grab".TON(IN := #_w1, PT := T#1S);
   "Green_Box_Pick&Place_TP_Grab".TP(IN := "Green_Box_Pick&Place_TON_Grab".Q, PT := T#4S);
   "Green_Box_PicknPlace_Grab" := "Green_Box_Pick&Place_TP_Grab".Q;
   "Green_Box_Pick&Place_TON_Z1".TON(IN := #_w1, PT := T#1S);
   "Green_Box_Pick&Place_TP_Z".TP(IN := "Green_Box_Pick&Place_TON_Z1".Q, PT := T#5S);
   "Green_Box_PicknPlace_Z" := "Green_Box_Pick&Place_TP_Z".Q AND NOT "Green_Box_Pick&Place_TON_Z2".Q;
   "Green_Box_Pick&Place_TON_Z2".TON(IN := "Green_Box_Pick&Place_TP_Z".Q AND NOT "Green_Box_Pick&Place_TON_Z3".Q,
                           PT := T#1S);
   "Green_Box_Pick&Place_TON_Z3".TON(IN := "Green_Box_Pick&Place_TP_Z".Q AND "Green_Box_Pick&Place_TON_Z2".Q,
                           PT := T#2S);
END_REGION

REGION Network 4
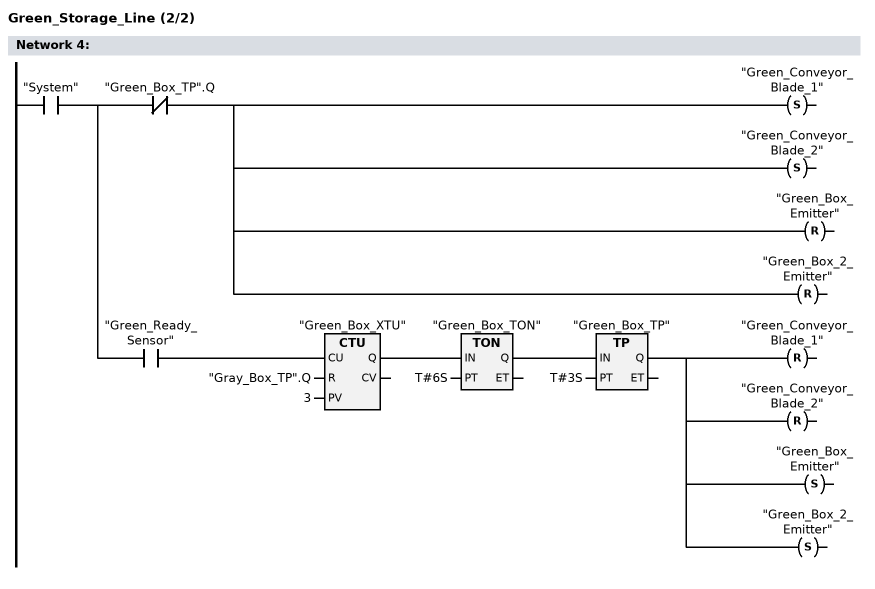
   IF "System" AND NOT "Green_Box_TP".Q THEN
       "Green_Conveyor_Blade_1" := TRUE;
       "Green_Conveyor_Blade_2" := TRUE;
       "Green_Box_Emitter" := FALSE;
       "Green_Box_2_Emitter" := FALSE;
   END_IF;
   "Green_Box_XTU".CTU(CU := "System" AND "Green_Ready_Sensor", R := "Gray_Box_TP".Q, PV := 3);
   "Green_Box_TON".TON(IN := "Green_Box_XTU".Q, PT := T#6S);
   "Green_Box_TP".TP(IN := "Green_Box_TON".Q, PT := T#3S);
   IF "Green_Box_TP".Q THEN
       "Green_Conveyor_Blade_1" := FALSE;
       "Green_Conveyor_Blade_2" := FALSE;
       "Green_Box_Emitter" := TRUE;
       "Green_Box_2_Emitter" := TRUE;
   END_IF;
END_REGION
END_FUNCTION_BLOCK

FUNCTION_BLOCK "Green_Store"   // FB9, LAD
{ S7_Optimized_Access := 'TRUE' }
VERSION : 0.1
   VAR_TEMP   // added for the SCL form of the ladder/FBD networks
      _w1 : Bool;
   END_VAR
BEGIN

REGION Network 1
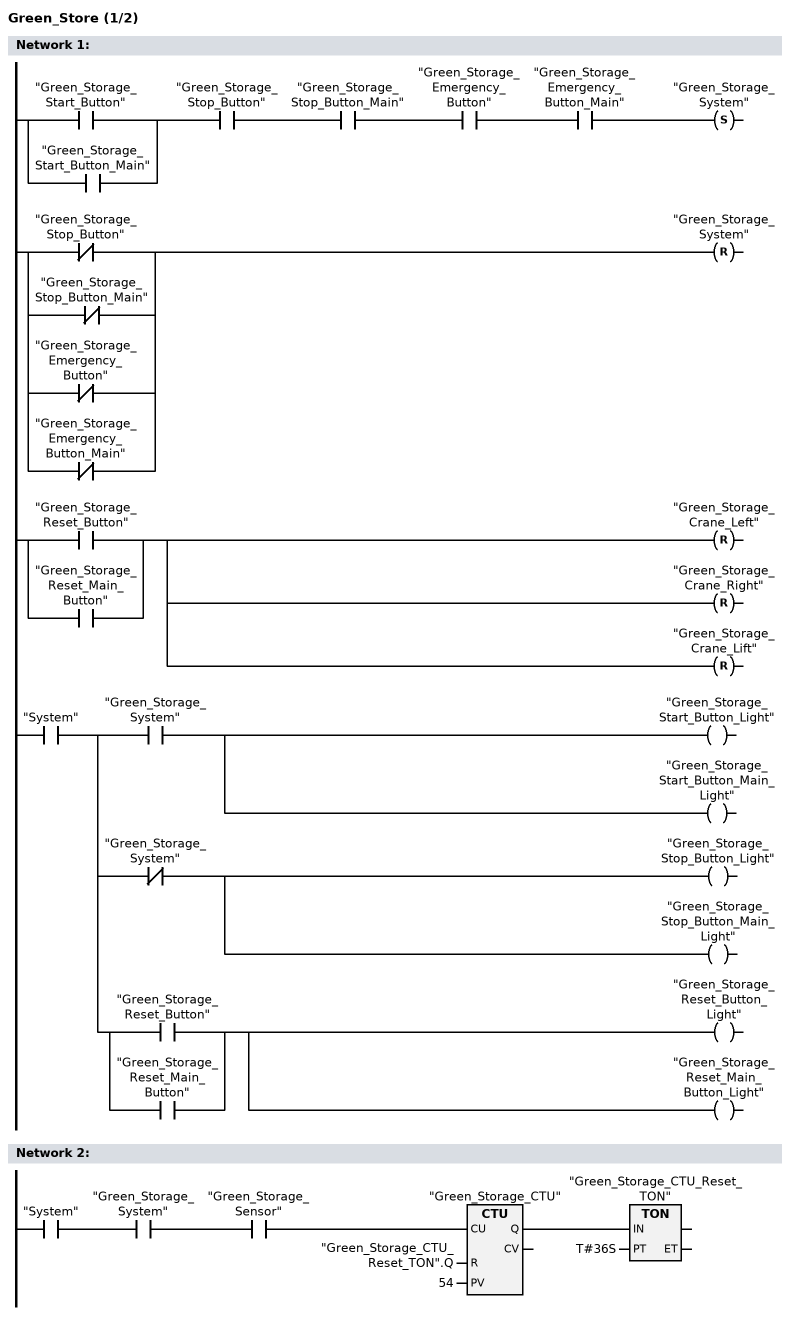
   RUNG wire#powerrail
      Contact( "Green_Storage_Start_Button" )
      wire#w1
      Contact( "Green_Storage_Stop_Button" )
      Contact( "Green_Storage_Stop_Button_Main" )
      Contact( "Green_Storage_Emergency_Button" )
      Contact( "Green_Storage_Emergency_Button_Main" )
      S_Coil( "Green_Storage_System" )
   END_RUNG
   RUNG wire#powerrail
      Contact( "Green_Storage_Start_Button_Main" )
   END_RUNG wire#w1
   RUNG wire#powerrail
      I_Contact( "Green_Storage_Stop_Button" )
      wire#w2
      R_Coil( "Green_Storage_System" )
   END_RUNG
   RUNG wire#powerrail
      I_Contact( "Green_Storage_Stop_Button_Main" )
   END_RUNG wire#w2
   RUNG wire#powerrail
      I_Contact( "Green_Storage_Emergency_Button" )
   END_RUNG wire#w2
   RUNG wire#powerrail
      I_Contact( "Green_Storage_Emergency_Button_Main" )
   END_RUNG wire#w2
   RUNG wire#powerrail
      Contact( "Green_Storage_Reset_Button" )
      wire#w3
      R_Coil( "Green_Storage_Crane_Left" )
   END_RUNG
   RUNG wire#powerrail
      Contact( "Green_Storage_Reset_Main_Button" )
   END_RUNG wire#w3
   RUNG wire#w3
      R_Coil( "Green_Storage_Crane_Right" )
   END_RUNG
   RUNG wire#w3
      R_Coil( "Green_Storage_Crane_Lift" )
   END_RUNG
   RUNG wire#powerrail
      Contact( "System" )
      wire#w4
      Contact( "Green_Storage_System" )
      wire#w5
      Coil( "Green_Storage_Start_Button_Light" )
   END_RUNG
   RUNG wire#w5
      Coil( "Green_Storage_Start_Button_Main_Light" )
   END_RUNG
   RUNG wire#w4
      I_Contact( "Green_Storage_System" )
      wire#w6
      Coil( "Green_Storage_Stop_Button_Light" )
   END_RUNG
   RUNG wire#w6
      Coil( "Green_Storage_Stop_Button_Main_Light" )
   END_RUNG
   RUNG wire#w4
      Contact( "Green_Storage_Reset_Button" )
      wire#w7
      Coil( "Green_Storage_Reset_Button_Light" )
   END_RUNG
   RUNG wire#w4
      Contact( "Green_Storage_Reset_Main_Button" )
   END_RUNG wire#w7
   RUNG wire#w7
      Coil( "Green_Storage_Reset_Main_Button_Light" )
   END_RUNG
   // the same network as SCL:
   IF ("Green_Storage_Start_Button" OR "Green_Storage_Start_Button_Main") AND "Green_Storage_Stop_Button" AND "Green_Storage_Stop_Button_Main" AND "Green_Storage_Emergency_Button" AND "Green_Storage_Emergency_Button_Main" THEN
       "Green_Storage_System" := TRUE;
   END_IF;
   IF NOT "Green_Storage_Stop_Button" OR NOT "Green_Storage_Stop_Button_Main" OR NOT "Green_Storage_Emergency_Button" OR NOT "Green_Storage_Emergency_Button_Main" THEN
       "Green_Storage_System" := FALSE;
   END_IF;
   IF "Green_Storage_Reset_Button" OR "Green_Storage_Reset_Main_Button" THEN
       "Green_Storage_Crane_Left" := FALSE;
       "Green_Storage_Crane_Right" := FALSE;
       "Green_Storage_Crane_Lift" := FALSE;
   END_IF;
   "Green_Storage_Start_Button_Light" := "System" AND "Green_Storage_System";
   "Green_Storage_Start_Button_Main_Light" := "Green_Storage_Start_Button_Light";
   "Green_Storage_Stop_Button_Light" := "System" AND NOT "Green_Storage_System";
   "Green_Storage_Stop_Button_Main_Light" := "Green_Storage_Stop_Button_Light";
   "Green_Storage_Reset_Button_Light" := "System" AND ("Green_Storage_Reset_Button" OR "Green_Storage_Reset_Main_Button");
   "Green_Storage_Reset_Main_Button_Light" := "Green_Storage_Reset_Button_Light";
END_REGION

REGION Network 2
   "Green_Storage_CTU".CTU(CU := "System" AND "Green_Storage_System" AND "Green_Storage_Sensor",
                           R := "Green_Storage_CTU_Reset_TON".Q,
                           PV := 54);
   "Green_Storage_CTU_Reset_TON".TON(IN := "Green_Storage_CTU".Q, PT := T#36S);
END_REGION

REGION Network 3
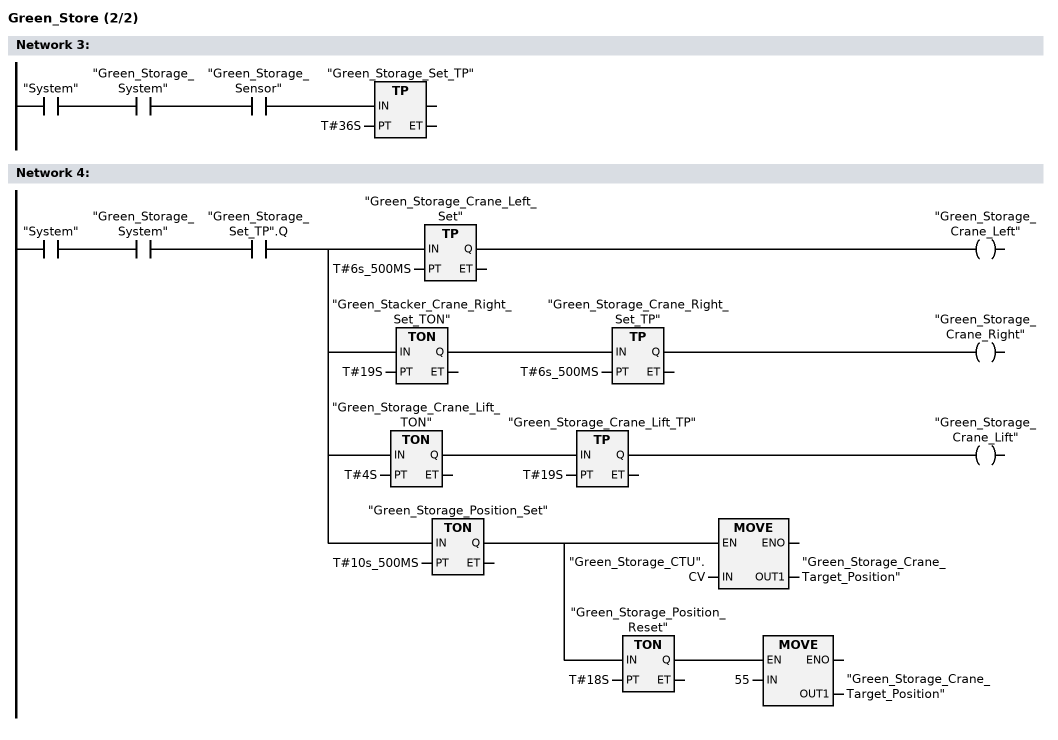
   "Green_Storage_Set_TP".TP(IN := "System" AND "Green_Storage_System" AND "Green_Storage_Sensor", PT := T#36S);
END_REGION

REGION Network 4
   #_w1 := "System" AND "Green_Storage_System" AND "Green_Storage_Set_TP".Q;
   "Green_Storage_Crane_Left_Set".TP(IN := #_w1, PT := T#6s_500MS);
   "Green_Storage_Crane_Left" := "Green_Storage_Crane_Left_Set".Q;
   "Green_Stacker_Crane_Right_Set_TON".TON(IN := #_w1, PT := T#19S);
   "Green_Storage_Crane_Right_Set_TP".TP(IN := "Green_Stacker_Crane_Right_Set_TON".Q, PT := T#6s_500MS);
   "Green_Storage_Crane_Right" := "Green_Storage_Crane_Right_Set_TP".Q;
   "Green_Storage_Crane_Lift_TON".TON(IN := #_w1, PT := T#4S);
   "Green_Storage_Crane_Lift_TP".TP(IN := "Green_Storage_Crane_Lift_TON".Q, PT := T#19S);
   "Green_Storage_Crane_Lift" := "Green_Storage_Crane_Lift_TP".Q;
   "Green_Storage_Position_Set".TON(IN := #_w1, PT := T#10s_500MS);
   IF "Green_Storage_Position_Set".Q THEN
       "Green_Storage_Crane_Target_Position" := "Green_Storage_CTU".CV;
   END_IF;
   "Green_Storage_Position_Reset".TON(IN := "Green_Storage_Position_Set".Q, PT := T#18S);
   IF "Green_Storage_Position_Reset".Q THEN "Green_Storage_Crane_Target_Position" := 55; END_IF;
END_REGION
END_FUNCTION_BLOCK

FUNCTION_BLOCK "MixingCorrector"   // FB10, LAD
{ S7_Optimized_Access := 'TRUE' }
VERSION : 0.1
BEGIN

REGION Network 1
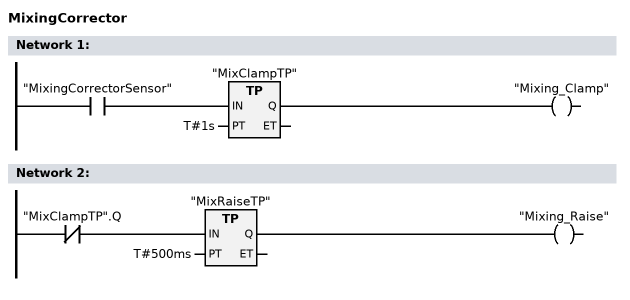
   "MixClampTP".TP(IN := "MixingCorrectorSensor", PT := T#1s);
   "Mixing_Clamp" := "MixClampTP".Q;
END_REGION

REGION Network 2
   "MixRaiseTP".TP(IN := NOT "MixClampTP".Q, PT := T#500ms);
   "Mixing_Raise" := "MixRaiseTP".Q;
END_REGION
END_FUNCTION_BLOCK

FUNCTION_BLOCK "BrandNewFill"   // FB12, LAD
{ S7_Optimized_Access := 'TRUE' }
VERSION : 0.1
BEGIN

REGION Network 1
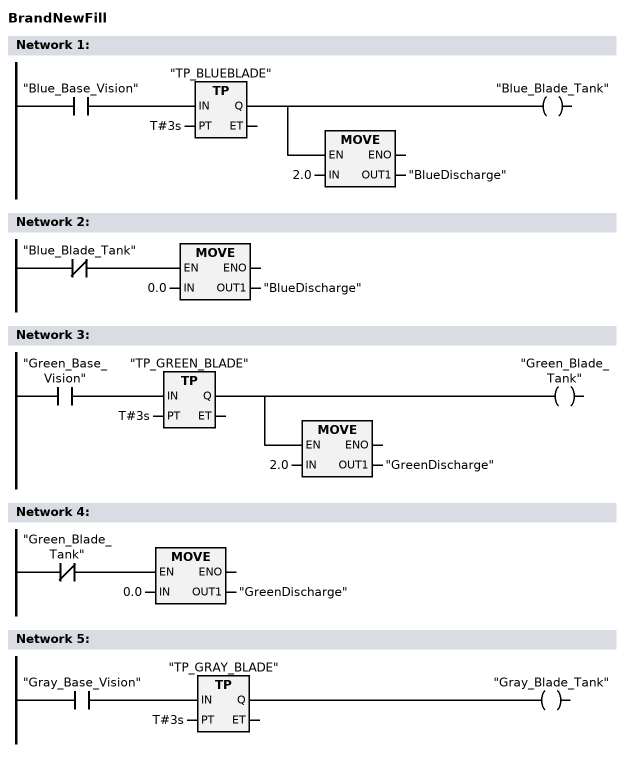
   "TP_BLUEBLADE".TP(IN := "Blue_Base_Vision", PT := T#3s);
   "Blue_Blade_Tank" := "TP_BLUEBLADE".Q;
   IF "TP_BLUEBLADE".Q THEN "BlueDischarge" := 2.0; END_IF;
END_REGION

REGION Network 2
   RUNG wire#powerrail
      I_Contact( "Blue_Blade_Tank" )
      Move(in := 0.0, out1 => "BlueDischarge")
   END_RUNG
   // the same network as SCL:
   IF NOT "Blue_Blade_Tank" THEN "BlueDischarge" := 0.0; END_IF;
END_REGION

REGION Network 3
   "TP_GREEN_BLADE".TP(IN := "Green_Base_Vision", PT := T#3s);
   "Green_Blade_Tank" := "TP_GREEN_BLADE".Q;
   IF "TP_GREEN_BLADE".Q THEN "GreenDischarge" := 2.0; END_IF;
END_REGION

REGION Network 4
   RUNG wire#powerrail
      I_Contact( "Green_Blade_Tank" )
      Move(in := 0.0, out1 => "GreenDischarge")
   END_RUNG
   // the same network as SCL:
   IF NOT "Green_Blade_Tank" THEN "GreenDischarge" := 0.0; END_IF;
END_REGION

REGION Network 5
   "TP_GRAY_BLADE".TP(IN := "Gray_Base_Vision", PT := T#3s);
   "Gray_Blade_Tank" := "TP_GRAY_BLADE".Q;
END_REGION
END_FUNCTION_BLOCK

FUNCTION "MHJ-PLC-Lab-Function-S71500" : Void   // FC9000, SCL
{ S7_Optimized_Access := 'TRUE' }
VERSION : 0.1
   VAR_TEMP
      Value : Byte;
      ForCounter : Int;
   END_VAR
   VAR CONSTANT
      Value_01_DW : DWord := 16#1223_5486;
      Value_02_DW : DWord := 16#A6C9_D1F5;
   END_VAR
BEGIN

   #Value:=PEEK(area := 16#82,
        dbNumber := 0,
        byteOffset := 511);
   #Value := #Value + 1;

   POKE(area := 16#82,
        dbNumber := 0,
        byteOffset := 511,
        value := #Value);

   POKE(area := 16#82,
        dbNumber := 0,
        byteOffset := 1016,
        value := #Value_01_DW);
   POKE(area := 16#82,
        dbNumber := 0,
        byteOffset := 1020,
        value := #Value_02_DW);

   FOR #ForCounter := 0 TO 63 DO
       #Value:=PEEK(area := 16#1,
            dbNumber := 0,
            byteOffset := #ForCounter);
       POKE(area := 16#81,
            dbNumber := 0,
            byteOffset := #ForCounter,
            value := #Value);
   END_FOR;
   #Value := PEEK(area := 16#1,
                  dbNumber := 0,
                  byteOffset := 512);
   POKE(area := 16#82,
        dbNumber := 0,
        byteOffset := 512,
        value := #Value);
END_FUNCTION

ORGANIZATION_BLOCK "Main"   // OB1, LAD, ProgramCycle
TITLE = "Main Program Sweep (Cycle)"
{ S7_Optimized_Access := 'TRUE' }
VERSION : 0.1
   VAR_INPUT
      Initial_Call : Bool;   // Initial call of this OB
      Remanence : Bool;   // =True, if remanent data are available
   END_VAR
BEGIN

REGION Network 1
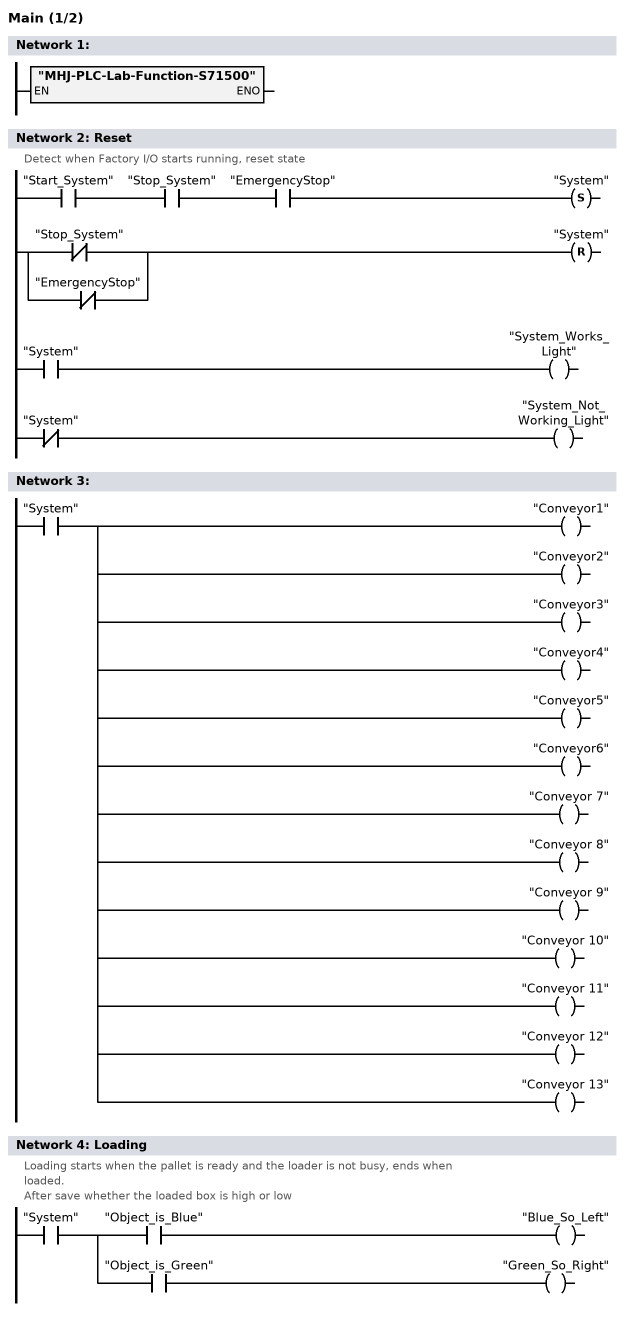
   RUNG wire#powerrail
      "MHJ-PLC-Lab-Function-S71500"()
   END_RUNG
   // the same network as SCL:
   "MHJ-PLC-Lab-Function-S71500"();
END_REGION

REGION Network 2: Reset
   // Detect when Factory I/O starts running, reset state
   RUNG wire#powerrail
      Contact( "Start_System" )
      Contact( "Stop_System" )
      Contact( "EmergencyStop" )
      S_Coil( "System" )
   END_RUNG
   RUNG wire#powerrail
      I_Contact( "Stop_System" )
      wire#w1
      R_Coil( "System" )
   END_RUNG
   RUNG wire#powerrail
      I_Contact( "EmergencyStop" )
   END_RUNG wire#w1
   RUNG wire#powerrail
      Contact( "System" )
      Coil( "System_Works_Light" )
   END_RUNG
   RUNG wire#powerrail
      I_Contact( "System" )
      Coil( "System_Not_Working_Light" )
   END_RUNG
   // the same network as SCL:
   IF "Start_System" AND "Stop_System" AND "EmergencyStop" THEN "System" := TRUE; END_IF;
   IF NOT "Stop_System" OR NOT "EmergencyStop" THEN "System" := FALSE; END_IF;
   "System_Works_Light" := "System";
   "System_Not_Working_Light" := NOT "System";
END_REGION

REGION Network 3
   RUNG wire#powerrail
      Contact( "System" )
      wire#w1
      Coil( "Conveyor1" )
   END_RUNG
   RUNG wire#w1
      Coil( "Conveyor2" )
   END_RUNG
   RUNG wire#w1
      Coil( "Conveyor3" )
   END_RUNG
   RUNG wire#w1
      Coil( "Conveyor4" )
   END_RUNG
   RUNG wire#w1
      Coil( "Conveyor5" )
   END_RUNG
   RUNG wire#w1
      Coil( "Conveyor6" )
   END_RUNG
   RUNG wire#w1
      Coil( "Conveyor 7" )
   END_RUNG
   RUNG wire#w1
      Coil( "Conveyor 8" )
   END_RUNG
   RUNG wire#w1
      Coil( "Conveyor 9" )
   END_RUNG
   RUNG wire#w1
      Coil( "Conveyor 10" )
   END_RUNG
   RUNG wire#w1
      Coil( "Conveyor 11" )
   END_RUNG
   RUNG wire#w1
      Coil( "Conveyor 12" )
   END_RUNG
   RUNG wire#w1
      Coil( "Conveyor 13" )
   END_RUNG
   // the same network as SCL:
   "Conveyor1" := "System";
   "Conveyor2" := "System";
   "Conveyor3" := "System";
   "Conveyor4" := "System";
   "Conveyor5" := "System";
   "Conveyor6" := "System";
   "Conveyor 7" := "System";
   "Conveyor 8" := "System";
   "Conveyor 9" := "System";
   "Conveyor 10" := "System";
   "Conveyor 11" := "System";
   "Conveyor 12" := "System";
   "Conveyor 13" := "System";
END_REGION

REGION Network 4: Loading
   // Loading starts when the pallet is ready and the loader is not busy, ends when 
   // loaded.
   // After save whether the loaded box is high or low
   RUNG wire#powerrail
      Contact( "System" )
      wire#w1
      Contact( "Object_is_Blue" )
      Coil( "Blue_So_Left" )
   END_RUNG
   RUNG wire#w1
      Contact( "Object_is_Green" )
      Coil( "Green_So_Right" )
   END_RUNG
   // the same network as SCL:
   "Blue_So_Left" := "System" AND "Object_is_Blue";
   "Green_So_Right" := "System" AND "Object_is_Green";
END_REGION

REGION Network 5
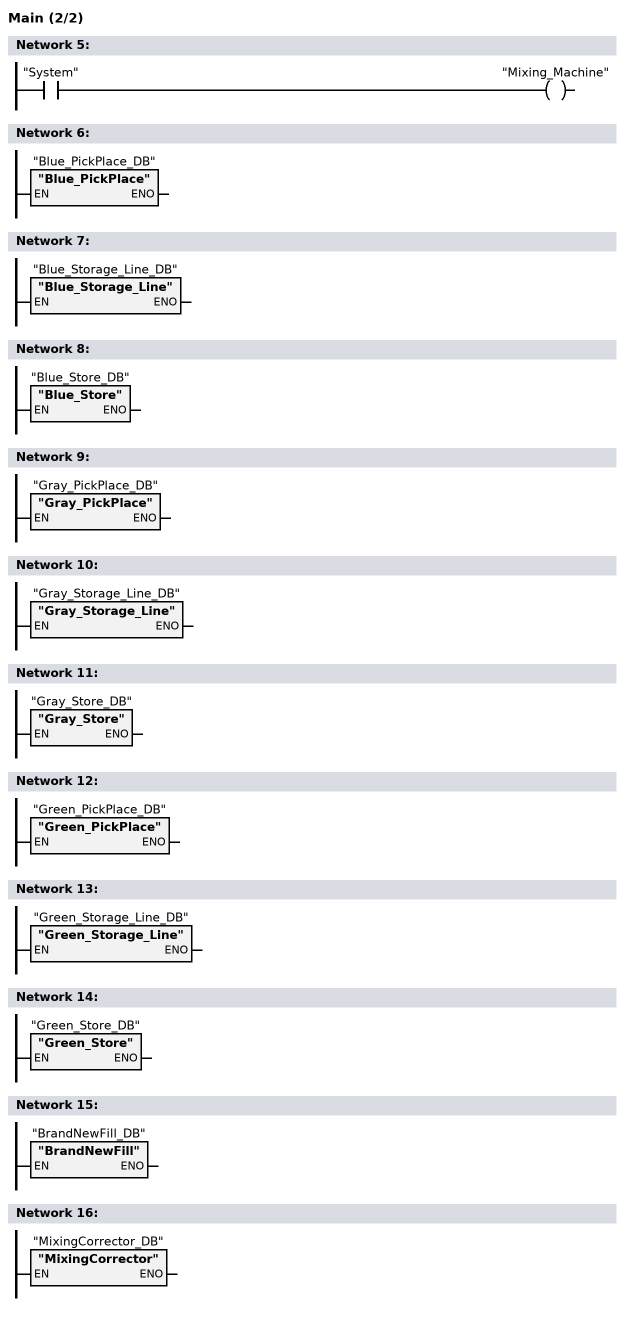
   RUNG wire#powerrail
      Contact( "System" )
      Coil( "Mixing_Machine" )
   END_RUNG
   // the same network as SCL:
   "Mixing_Machine" := "System";
END_REGION

REGION Network 6
   RUNG wire#powerrail
      "Blue_PickPlace_DB"()
   END_RUNG
   // the same network as SCL:
   "Blue_PickPlace_DB"();   // "Blue_PickPlace"
END_REGION

REGION Network 7
   RUNG wire#powerrail
      "Blue_Storage_Line_DB"()
   END_RUNG
   // the same network as SCL:
   "Blue_Storage_Line_DB"();   // "Blue_Storage_Line"
END_REGION

REGION Network 8
   RUNG wire#powerrail
      "Blue_Store_DB"()
   END_RUNG
   // the same network as SCL:
   "Blue_Store_DB"();   // "Blue_Store"
END_REGION

REGION Network 9
   RUNG wire#powerrail
      "Gray_PickPlace_DB"()
   END_RUNG
   // the same network as SCL:
   "Gray_PickPlace_DB"();   // "Gray_PickPlace"
END_REGION

REGION Network 10
   RUNG wire#powerrail
      "Gray_Storage_Line_DB"()
   END_RUNG
   // the same network as SCL:
   "Gray_Storage_Line_DB"();   // "Gray_Storage_Line"
END_REGION

REGION Network 11
   RUNG wire#powerrail
      "Gray_Store_DB"()
   END_RUNG
   // the same network as SCL:
   "Gray_Store_DB"();   // "Gray_Store"
END_REGION

REGION Network 12
   RUNG wire#powerrail
      "Green_PickPlace_DB"()
   END_RUNG
   // the same network as SCL:
   "Green_PickPlace_DB"();   // "Green_PickPlace"
END_REGION

REGION Network 13
   RUNG wire#powerrail
      "Green_Storage_Line_DB"()
   END_RUNG
   // the same network as SCL:
   "Green_Storage_Line_DB"();   // "Green_Storage_Line"
END_REGION

REGION Network 14
   RUNG wire#powerrail
      "Green_Store_DB"()
   END_RUNG
   // the same network as SCL:
   "Green_Store_DB"();   // "Green_Store"
END_REGION

REGION Network 15
   RUNG wire#powerrail
      "BrandNewFill_DB"()
   END_RUNG
   // the same network as SCL:
   "BrandNewFill_DB"();   // "BrandNewFill"
END_REGION

REGION Network 16
   RUNG wire#powerrail
      "MixingCorrector_DB"()
   END_RUNG
   // the same network as SCL:
   "MixingCorrector_DB"();   // "MixingCorrector"
END_REGION
END_ORGANIZATION_BLOCK

ORGANIZATION_BLOCK "Blue_PID"   // OB30, LAD, CyclicInterrupt
{ S7_Optimized_Access := 'TRUE' }
VERSION : 0.1
   VAR_INPUT
      Initial_Call : Bool;   // Initial call of this OB
      Event_Count : Int;   // Events discarded
   END_VAR
BEGIN

REGION Network 1
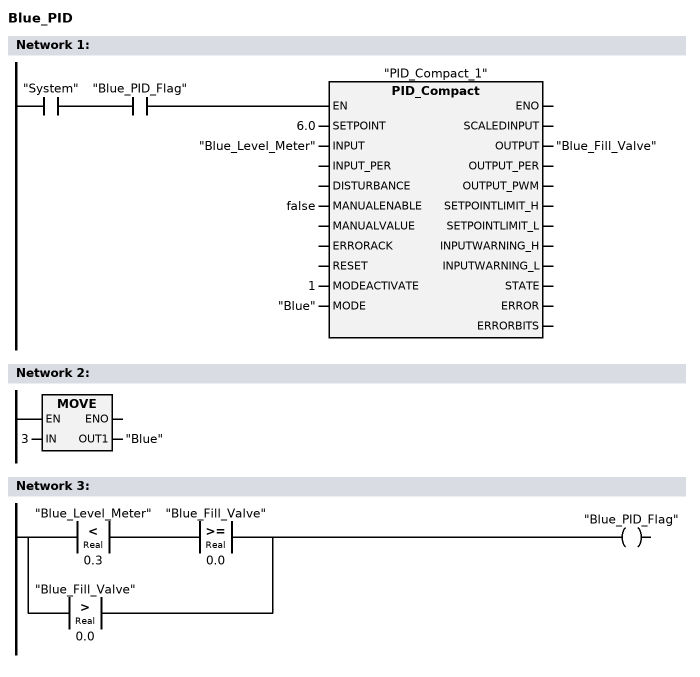
   IF "System" AND "Blue_PID_Flag" THEN
       "PID_Compact_1"(Setpoint := 6.0,   // PID_Compact
                       Input := "Blue_Level_Meter",
                       ManualEnable := false,
                       ModeActivate := 1,
                       Mode := "Blue",
                       Output => "Blue_Fill_Valve");
   END_IF;
END_REGION

REGION Network 2
   RUNG wire#powerrail
      Move(in := 3, out1 => "Blue")
   END_RUNG
   // the same network as SCL:
   "Blue" := 3;
END_REGION

REGION Network 3
   RUNG wire#powerrail
      { S7_Templates := "SrcType := Real" } LT_Contact(in1 := "Blue_Level_Meter", in2 := 0.3)
      { S7_Templates := "SrcType := Real" } GE_Contact(in1 := "Blue_Fill_Valve", in2 := 0.0)
      wire#w1
      Coil( "Blue_PID_Flag" )
   END_RUNG
   RUNG wire#powerrail
      { S7_Templates := "SrcType := Real" } GT_Contact(in1 := "Blue_Fill_Valve", in2 := 0.0)
   END_RUNG wire#w1
   // the same network as SCL:
   "Blue_PID_Flag" := (("Blue_Level_Meter" < 0.3) AND ("Blue_Fill_Valve" >= 0.0)) OR ("Blue_Fill_Valve" > 0.0);
END_REGION
END_ORGANIZATION_BLOCK

ORGANIZATION_BLOCK "Green_PID"   // OB31, LAD, CyclicInterrupt
{ S7_Optimized_Access := 'TRUE' }
VERSION : 0.1
   VAR_INPUT
      Initial_Call : Bool;   // Initial call of this OB
      Event_Count : Int;   // Events discarded
   END_VAR
BEGIN

REGION Network 1
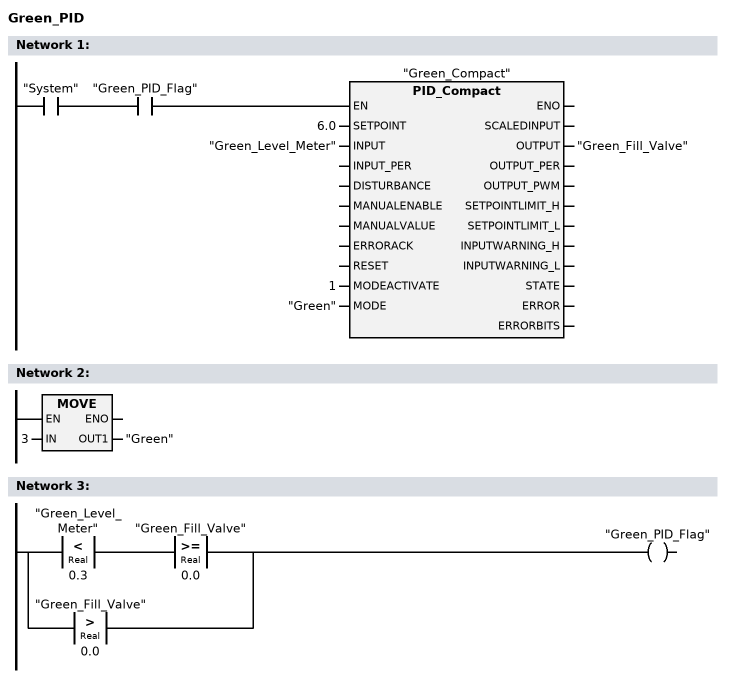
   IF "System" AND "Green_PID_Flag" THEN
       "Green_Compact"(Setpoint := 6.0,   // PID_Compact
                       Input := "Green_Level_Meter",
                       ModeActivate := 1,
                       Mode := "Green",
                       Output => "Green_Fill_Valve");
   END_IF;
END_REGION

REGION Network 2
   RUNG wire#powerrail
      Move(in := 3, out1 => "Green")
   END_RUNG
   // the same network as SCL:
   "Green" := 3;
END_REGION

REGION Network 3
   RUNG wire#powerrail
      { S7_Templates := "SrcType := Real" } LT_Contact(in1 := "Green_Level_Meter", in2 := 0.3)
      { S7_Templates := "SrcType := Real" } GE_Contact(in1 := "Green_Fill_Valve", in2 := 0.0)
      wire#w1
      Coil( "Green_PID_Flag" )
   END_RUNG
   RUNG wire#powerrail
      { S7_Templates := "SrcType := Real" } GT_Contact(in1 := "Green_Fill_Valve", in2 := 0.0)
   END_RUNG wire#w1
   // the same network as SCL:
   "Green_PID_Flag" := (("Green_Level_Meter" < 0.3) AND ("Green_Fill_Valve" >= 0.0)) OR ("Green_Fill_Valve" > 0.0);
END_REGION
END_ORGANIZATION_BLOCK

ORGANIZATION_BLOCK "Gray_PID"   // OB32, LAD, CyclicInterrupt
{ S7_Optimized_Access := 'TRUE' }
VERSION : 0.1
   VAR_INPUT
      Initial_Call : Bool;   // Initial call of this OB
      Event_Count : Int;   // Events discarded
   END_VAR
BEGIN

REGION Network 1
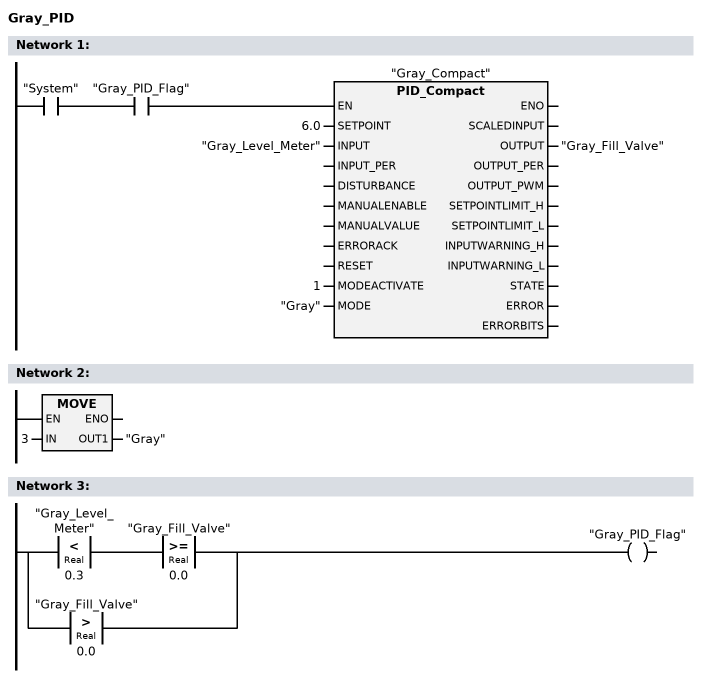
   IF "System" AND "Gray_PID_Flag" THEN
       "Gray_Compact"(Setpoint := 6.0,   // PID_Compact
                      Input := "Gray_Level_Meter",
                      ModeActivate := 1,
                      Mode := "Gray",
                      Output => "Gray_Fill_Valve");
   END_IF;
END_REGION

REGION Network 2
   RUNG wire#powerrail
      Move(in := 3, out1 => "Gray")
   END_RUNG
   // the same network as SCL:
   "Gray" := 3;
END_REGION

REGION Network 3
   RUNG wire#powerrail
      { S7_Templates := "SrcType := Real" } LT_Contact(in1 := "Gray_Level_Meter", in2 := 0.3)
      { S7_Templates := "SrcType := Real" } GE_Contact(in1 := "Gray_Fill_Valve", in2 := 0.0)
      wire#w1
      Coil( "Gray_PID_Flag" )
   END_RUNG
   RUNG wire#powerrail
      { S7_Templates := "SrcType := Real" } GT_Contact(in1 := "Gray_Fill_Valve", in2 := 0.0)
   END_RUNG wire#w1
   // the same network as SCL:
   "Gray_PID_Flag" := (("Gray_Level_Meter" < 0.3) AND ("Gray_Fill_Valve" >= 0.0)) OR ("Gray_Fill_Valve" > 0.0);
END_REGION
END_ORGANIZATION_BLOCK

ORGANIZATION_BLOCK "Emitter"   // OB33, LAD, CyclicInterrupt
{ S7_Optimized_Access := 'TRUE' }
VERSION : 0.1
   VAR_INPUT
      Initial_Call : Bool;   // Initial call of this OB
      Event_Count : Int;   // Events discarded
   END_VAR
BEGIN

REGION Network 1
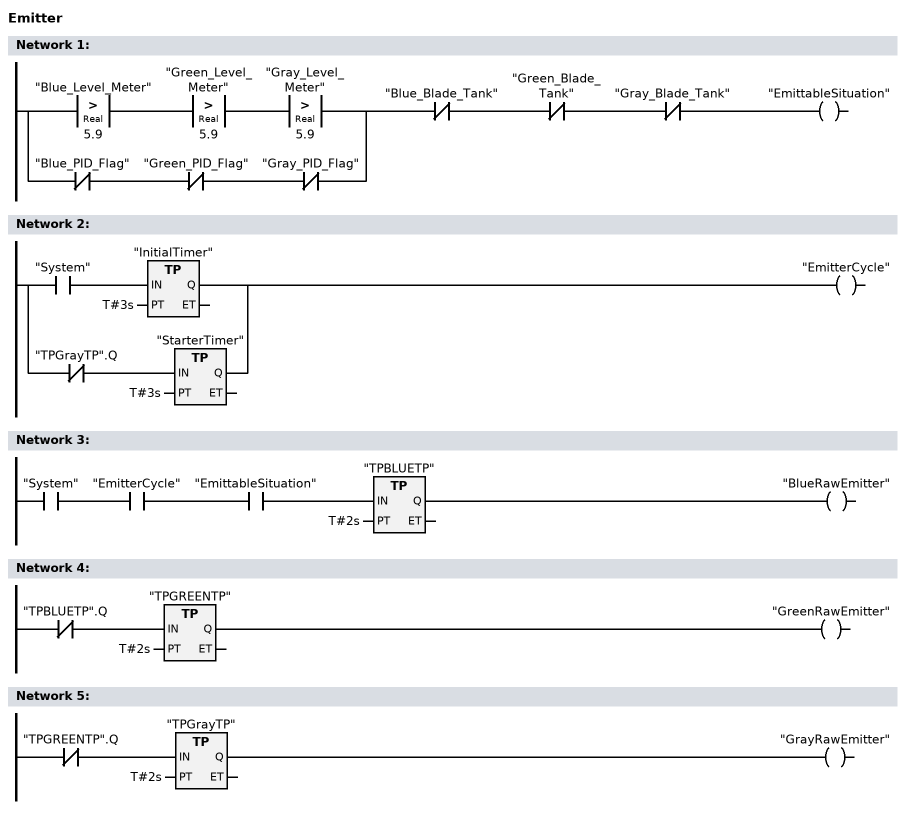
   RUNG wire#powerrail
      { S7_Templates := "SrcType := Real" } GT_Contact(in1 := "Blue_Level_Meter", in2 := 5.9)
      { S7_Templates := "SrcType := Real" } GT_Contact(in1 := "Green_Level_Meter", in2 := 5.9)
      { S7_Templates := "SrcType := Real" } GT_Contact(in1 := "Gray_Level_Meter", in2 := 5.9)
      wire#w1
      I_Contact( "Blue_Blade_Tank" )
      I_Contact( "Green_Blade_Tank" )
      I_Contact( "Gray_Blade_Tank" )
      Coil( "EmittableSituation" )
   END_RUNG
   RUNG wire#powerrail
      I_Contact( "Blue_PID_Flag" )
      I_Contact( "Green_PID_Flag" )
      I_Contact( "Gray_PID_Flag" )
   END_RUNG wire#w1
   // the same network as SCL:
   "EmittableSituation" := ((("Blue_Level_Meter" > 5.9) AND ("Green_Level_Meter" > 5.9) AND ("Gray_Level_Meter" > 5.9)) OR (NOT "Blue_PID_Flag" AND NOT "Green_PID_Flag" AND NOT "Gray_PID_Flag")) AND NOT "Blue_Blade_Tank" AND NOT "Green_Blade_Tank" AND NOT "Gray_Blade_Tank";
END_REGION

REGION Network 2
   "InitialTimer".TP(IN := "System", PT := T#3s);
   "StarterTimer".TP(IN := NOT "TPGrayTP".Q, PT := T#3s);
   "EmitterCycle" := "InitialTimer".Q OR "StarterTimer".Q;
END_REGION

REGION Network 3
   "TPBLUETP".TP(IN := "System" AND "EmitterCycle" AND "EmittableSituation", PT := T#2s);
   "BlueRawEmitter" := "TPBLUETP".Q;
END_REGION

REGION Network 4
   "TPGREENTP".TP(IN := NOT "TPBLUETP".Q, PT := T#2s);
   "GreenRawEmitter" := "TPGREENTP".Q;
END_REGION

REGION Network 5
   "TPGrayTP".TP(IN := NOT "TPGREENTP".Q, PT := T#2s);
   "GrayRawEmitter" := "TPGrayTP".Q;
END_REGION
END_ORGANIZATION_BLOCK